KUKA KRL program: Machining3.src

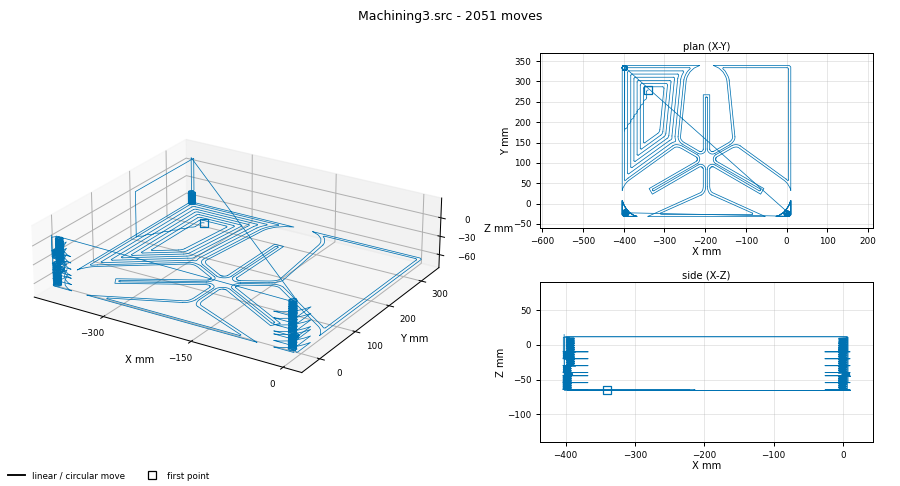
[picture p0: tool path of Machining3.src, 2051 of 2051 moves have a stored position in this frame; points joined in program order, loops and branches not executed]
&ACCESS RVP
&REL 1
&PARAM TEMPLATE = C:\KRC\Roboter\Template\vorgabe
&PARAM EDITMASK = *
DEF Machining3 ( )
LIN {X -339.907,Y 279.175,Z -64.500,A 0.015,B 0.000,C 180.000} C_DIS
CIRC {X -342.631,Y 278.046,Z -64.500,A 0.015,B -0.000,C -180.000},{X -343.760,Y 275.322,Z -64.500,A 0.015,B -0.000,C -180.000} C_DIS
LIN {X -343.759,Y 260.861,Z -64.500,A 0.015,B 0.000,C 180.000} C_DIS
CIRC {X -344.825,Y 257.341,Z -64.500,A 0.015,B 0.000,C 180.000},{X -347.664,Y 255.003,Z -64.500,A 0.015,B -0.000,C -180.000} C_DIS
CIRC {X -350.503,Y 252.666,Z -64.500,A 0.015,B 0.000,C 180.000},{X -351.569,Y 249.146,Z -64.500,A 0.015,B 0.000,C -180.000} C_DIS
LIN {X -351.566,Y 151.241,Z -64.500,A 0.015,B 0.000,C 180.000} C_DIS
CIRC {X -350.453,Y 149.418,Z -64.500,A 0.015,B 0.000,C -180.000},{X -348.323,Y 149.578,Z -64.500,A 0.015,B -0.000,C -180.000} C_DIS
LIN {X -316.688,Y 172.314,Z -64.500,A 0.015,B 0.000,C 180.000} C_DIS
CIRC {X -313.049,Y 176.334,Z -64.500,A 0.015,B 0.000,C 180.000},{X -311.385,Y 181.496,Z -64.500,A 0.015,B 0.000,C 180.000} C_DIS
LIN {X -301.199,Y 283.221,Z -64.500,A 0.015,B 0.000,C 180.000} C_DIS
CIRC {X -302.067,Y 285.859,Z -64.500,A 0.015,B 0.000,C 180.000},{X -304.605,Y 286.985,Z -64.500,A 0.015,B 0.000,C 180.000} C_DIS
LIN {X -347.717,Y 286.984,Z -64.500,A 0.015,B 0.000,C 180.000} C_DIS
CIRC {X -350.441,Y 285.856,Z -64.500,A 0.015,B 0.000,C 180.000},{X -351.570,Y 283.131,Z -64.500,A 0.015,B 0.000,C 180.000} C_DIS
LIN {X -351.569,Y 249.146,Z -64.500,A 0.015,B 0.000,C 180.000} C_DIS
CIRC {X -352.634,Y 245.626,Z -64.500,A 0.015,B 0.000,C 180.000},{X -355.473,Y 243.289,Z -64.500,A 0.015,B 0.000,C -180.000} C_DIS
CIRC {X -358.312,Y 240.951,Z -64.500,A 0.015,B 0.000,C 180.000},{X -359.378,Y 237.431,Z -64.500,A 0.015,B 0.000,C -180.000} C_DIS
LIN {X -359.375,Y 136.010,Z -64.500,A 0.015,B -0.000,C 180.000} C_DIS
CIRC {X -358.262,Y 134.188,Z -64.500,A 0.015,B 0.000,C 180.000},{X -356.132,Y 134.348,Z -64.500,A 0.015,B 0.000,C 180.000} C_DIS
LIN {X -309.268,Y 168.029,Z -64.500,A 0.015,B 0.000,C 180.000} C_DIS
CIRC {X -305.629,Y 172.049,Z -64.500,A 0.015,B 0.000,C -180.000},{X -303.966,Y 177.211,Z -64.500,A 0.015,B 0.000,C -180.000} C_DIS
LIN {X -292.568,Y 291.031,Z -64.500,A 0.015,B 0.000,C 180.000} C_DIS
CIRC {X -293.436,Y 293.669,Z -64.500,A 0.015,B -0.000,C -180.000},{X -295.974,Y 294.795,Z -64.500,A 0.015,B 0.000,C 180.000} C_DIS
LIN {X -355.527,Y 294.794,Z -64.500,A 0.015,B -0.000,C -180.000} C_DIS
CIRC {X -358.251,Y 293.665,Z -64.500,A 0.015,B 0.000,C -180.000},{X -359.380,Y 290.941,Z -64.500,A 0.015,B 0.000,C -180.000} C_DIS
LIN {X -359.378,Y 237.431,Z -64.500,A 0.015,B 0.000,C 180.000} C_DIS
CIRC {X -360.444,Y 233.911,Z -64.500,A 0.015,B 0.000,C 180.000},{X -363.283,Y 231.574,Z -64.500,A 0.015,B 0.000,C -180.000} C_DIS
CIRC {X -366.122,Y 229.236,Z -64.500,A 0.015,B 0.000,C -180.000},{X -367.188,Y 225.716,Z -64.500,A 0.015,B 0.000,C -180.000} C_DIS
LIN {X -367.185,Y 120.780,Z -64.500,A 0.015,B 0.000,C 180.000} C_DIS
CIRC {X -366.071,Y 118.958,Z -64.500,A 0.015,B -0.000,C 180.000},{X -363.942,Y 119.117,Z -64.500,A 0.015,B 0.000,C 180.000} C_DIS
LIN {X -301.848,Y 163.744,Z -64.500,A 0.015,B 0.000,C -180.000} C_DIS
CIRC {X -298.209,Y 167.764,Z -64.500,A 0.015,B 0.000,C 180.000},{X -296.546,Y 172.925,Z -64.500,A 0.015,B -0.000,C 180.000} C_DIS
LIN {X -283.937,Y 298.841,Z -64.500,A 0.015,B 0.000,C -180.000} C_DIS
CIRC {X -284.805,Y 301.479,Z -64.500,A 0.015,B 0.000,C 180.000},{X -287.343,Y 302.605,Z -64.500,A 0.015,B 0.000,C 180.000} C_DIS
LIN {X -363.337,Y 302.603,Z -64.500,A 0.015,B 0.000,C -180.000} C_DIS
CIRC {X -366.061,Y 301.475,Z -64.500,A 0.015,B 0.000,C 180.000},{X -367.190,Y 298.750,Z -64.500,A 0.015,B 0.000,C -180.000} C_DIS
LIN {X -367.188,Y 225.716,Z -64.500,A 0.015,B 0.000,C 180.000} C_DIS
CIRC {X -368.253,Y 222.196,Z -64.500,A 0.015,B 0.000,C -180.000},{X -371.092,Y 219.859,Z -64.500,A 0.015,B -0.000,C 180.000} C_DIS
CIRC {X -373.931,Y 217.521,Z -64.500,A 0.015,B -0.000,C 180.000},{X -374.997,Y 214.001,Z -64.500,A 0.015,B -0.000,C -180.000} C_DIS
LIN {X -374.994,Y 105.550,Z -64.500,A 0.015,B 0.000,C 180.000} C_DIS
CIRC {X -373.881,Y 103.728,Z -64.500,A 0.015,B 0.000,C 180.000},{X -371.751,Y 103.887,Z -64.500,A 0.015,B 0.000,C 180.000} C_DIS
LIN {X -293.623,Y 160.038,Z -64.500,A 0.015,B 0.000,C 180.000} C_DIS
CIRC {X -290.605,Y 163.373,Z -64.500,A 0.015,B 0.000,C 180.000},{X -289.225,Y 167.654,Z -64.500,A 0.015,B 0.000,C -180.000} C_DIS
LIN {X -275.691,Y 303.585,Z -64.500,A 0.015,B 0.000,C -180.000} C_DIS
CIRC {X -275.563,Y 304.401,Z -64.500,A 0.015,B 0.000,C -180.000},{X -275.412,Y 305.213,Z -64.500,A 0.015,B 0.000,C 180.000} C_DIS
CIRC {X -275.258,Y 306.024,Z -64.500,A 0.015,B 0.000,C 180.000},{X -275.124,Y 306.839,Z -64.500,A 0.015,B 0.000,C 180.000} C_DIS
CIRC {X -275.837,Y 309.333,Z -64.500,A 0.015,B 0.000,C 180.000},{X -278.194,Y 310.415,Z -64.500,A 0.015,B -0.000,C 180.000} C_DIS
LIN {X -371.147,Y 310.413,Z -64.500,A 0.015,B 0.000,C 180.000} C_DIS
CIRC {X -373.871,Y 309.285,Z -64.500,A 0.015,B -0.000,C 180.000},{X -375.000,Y 306.560,Z -64.500,A 0.015,B -0.000,C -180.000} C_DIS
LIN {X -374.997,Y 214.001,Z -64.500,A 0.015,B 0.000,C 180.000} C_DIS
CIRC {X -376.063,Y 210.481,Z -64.500,A 0.015,B 0.000,C -180.000},{X -378.902,Y 208.144,Z -64.500,A 0.015,B -0.000,C 180.000} C_DIS
CIRC {X -381.741,Y 205.806,Z -64.500,A 0.015,B 0.000,C -180.000},{X -382.807,Y 202.286,Z -64.500,A 0.015,B -0.000,C -180.000} C_DIS
LIN {X -382.803,Y 90.320,Z -64.500,A 0.015,B 0.000,C 180.000} C_DIS
CIRC {X -381.690,Y 88.498,Z -64.500,A 0.015,B -0.000,C -180.000},{X -379.561,Y 88.657,Z -64.500,A 0.015,B -0.000,C -180.000} C_DIS
LIN {X -288.345,Y 154.359,Z -64.500,A 0.015,B 0.000,C -180.000} C_DIS
CIRC {X -287.556,Y 154.885,Z -64.500,A 0.015,B 0.000,C 180.000},{X -286.733,Y 155.355,Z -64.500,A 0.015,B 0.000,C 180.000} C_DIS
CIRC {X -285.893,Y 155.792,Z -64.500,A 0.015,B 0.000,C 180.000},{X -285.049,Y 156.222,Z -64.500,A 0.015,B 0.000,C 180.000} C_DIS
CIRC {X -282.420,Y 158.717,Z -64.500,A 0.015,B -0.000,C 180.000},{X -281.597,Y 162.247,Z -64.500,A 0.015,B 0.000,C -180.000} C_DIS
CIRC {X -281.654,Y 163.235,Z -64.500,A 0.015,B 0.000,C -180.000},{X -281.701,Y 164.223,Z -64.500,A 0.015,B 0.000,C 180.000} C_DIS
CIRC {X -281.709,Y 165.212,Z -64.500,A 0.015,B 0.000,C -180.000},{X -281.645,Y 166.200,Z -64.500,A 0.015,B -0.000,C 180.000} C_DIS
LIN {X -267.342,Y 307.304,Z -64.500,A 0.015,B 0.000,C -180.000} C_DIS
CIRC {X -266.874,Y 309.190,Z -64.500,A 0.015,B 0.000,C 180.000},{X -266.314,Y 311.051,Z -64.500,A 0.015,B 0.000,C 180.000} C_DIS
CIRC {X -265.723,Y 312.902,Z -64.500,A 0.015,B -0.000,C 180.000},{X -265.158,Y 314.761,Z -64.500,A 0.015,B 0.000,C 180.000} C_DIS
CIRC {X -265.585,Y 317.142,Z -64.500,A 0.015,B -0.000,C 180.000},{X -267.747,Y 318.225,Z -64.500,A 0.015,B -0.000,C -180.000} C_DIS
LIN {X -378.957,Y 318.223,Z -64.500,A 0.015,B 0.000,C 180.000} C_DIS
CIRC {X -381.681,Y 317.094,Z -64.500,A 0.015,B 0.000,C 180.000},{X -382.810,Y 314.370,Z -64.500,A 0.015,B -0.000,C 180.000} C_DIS
LIN {X -382.807,Y 202.286,Z -64.500,A 0.015,B -0.000,C 180.000} C_DIS
CIRC {X -383.872,Y 198.767,Z -64.500,A 0.015,B 0.000,C 180.000},{X -386.711,Y 196.429,Z -64.500,A 0.015,B 0.000,C -180.000} C_DIS
CIRC {X -389.550,Y 194.091,Z -64.500,A 0.015,B -0.000,C 180.000},{X -390.616,Y 190.572,Z -64.500,A 0.015,B 0.000,C 180.000} C_DIS
LIN {X -390.613,Y 75.090,Z -64.500,A 0.015,B 0.000,C -180.000} C_DIS
CIRC {X -389.499,Y 73.268,Z -64.500,A 0.015,B -0.000,C -180.000},{X -387.370,Y 73.427,Z -64.500,A 0.015,B 0.000,C -180.000} C_DIS
LIN {X -283.893,Y 148.164,Z -64.500,A 0.015,B 0.000,C 180.000} C_DIS
CIRC {X -281.828,Y 149.430,Z -64.500,A 0.015,B 0.000,C 180.000},{X -279.602,Y 150.381,Z -64.500,A 0.015,B 0.000,C -180.000} C_DIS
CIRC {X -277.293,Y 151.093,Z -64.500,A 0.015,B 0.000,C 180.000},{X -274.944,Y 151.659,Z -64.500,A 0.015,B 0.000,C 180.000} C_DIS
CIRC {X -272.900,Y 153.122,Z -64.500,A 0.015,B 0.000,C 180.000},{X -272.606,Y 155.618,Z -64.500,A 0.015,B -0.000,C -180.000} C_DIS
CIRC {X -273.087,Y 157.304,Z -64.500,A 0.015,B 0.000,C -180.000},{X -273.496,Y 159.009,Z -64.500,A 0.015,B 0.000,C 180.000} C_DIS
CIRC {X -273.810,Y 160.735,Z -64.500,A 0.015,B 0.000,C 180.000},{X -274.004,Y 162.478,Z -64.500,A 0.015,B 0.000,C 180.000} C_DIS
CIRC {X -274.055,Y 163.218,Z -64.500,A 0.015,B 0.000,C -180.000},{X -274.097,Y 163.958,Z -64.500,A 0.015,B 0.000,C 180.000} C_DIS
CIRC {X -274.106,Y 164.700,Z -64.500,A 0.015,B 0.000,C -180.000},{X -274.060,Y 165.440,Z -64.500,A 0.015,B 0.000,C 180.000} C_DIS
LIN {X -260.011,Y 305.675,Z -64.500,A 0.015,B 0.000,C -180.000} C_DIS
CIRC {X -259.128,Y 309.215,Z -64.500,A 0.015,B 0.000,C 180.000},{X -258.064,Y 312.705,Z -64.500,A 0.015,B -0.000,C 180.000} C_DIS
CIRC {X -256.737,Y 316.107,Z -64.500,A 0.015,B 0.000,C 180.000},{X -255.075,Y 319.359,Z -64.500,A 0.015,B -0.000,C 180.000} C_DIS
CIRC {X -254.574,Y 320.199,Z -64.500,A 0.015,B 0.000,C -180.000},{X -254.046,Y 321.023,Z -64.500,A 0.015,B -0.000,C -180.000} C_DIS
CIRC {X -253.518,Y 321.847,Z -64.500,A 0.015,B 0.000,C 180.000},{X -253.017,Y 322.687,Z -64.500,A 0.015,B 0.000,C -180.000} C_DIS
CIRC {X -253.018,Y 324.920,Z -64.500,A 0.015,B 0.000,C 180.000},{X -254.952,Y 326.036,Z -64.500,A 0.015,B 0.000,C 180.000} C_DIS
LIN {X -386.767,Y 326.032,Z -64.500,A 0.015,B 0.000,C 180.000} C_DIS
CIRC {X -389.491,Y 324.904,Z -64.500,A 0.015,B 0.000,C 180.000},{X -390.620,Y 322.179,Z -64.500,A 0.015,B 0.000,C 180.000} C_DIS
LIN {X -390.616,Y 190.572,Z -64.500,A 0.015,B -0.000,C 180.000} C_DIS
CIRC {X -391.682,Y 187.052,Z -64.500,A 0.015,B 0.000,C -180.000},{X -394.521,Y 184.714,Z -64.500,A 0.015,B 0.000,C 180.000} C_DIS
CIRC {X -397.360,Y 182.376,Z -64.500,A 0.015,B 0.000,C -180.000},{X -398.426,Y 178.857,Z -64.500,A 0.015,B 0.000,C -180.000} C_DIS
LIN {X -398.422,Y 58.563,Z -64.500,A 0.015,B -0.000,C 180.000} C_DIS
CIRC {X -397.348,Y 56.920,Z -64.500,A 0.015,B 0.000,C -180.000},{X -395.413,Y 57.247,Z -64.500,A 0.015,B 0.000,C 180.000} C_DIS
CIRC {X -393.893,Y 58.674,Z -64.500,A 0.015,B 0.000,C 180.000},{X -392.395,Y 60.124,Z -64.500,A 0.015,B -0.000,C 180.000} C_DIS
CIRC {X -390.853,Y 61.528,Z -64.500,A 0.015,B 0.000,C 180.000},{X -389.207,Y 62.809,Z -64.500,A 0.015,B 0.000,C -180.000} C_DIS
LIN {X -279.477,Y 142.021,Z -64.500,A 0.015,B 0.000,C 180.000} C_DIS
CIRC {X -274.513,Y 144.373,Z -64.500,A 0.015,B 0.000,C 180.000},{X -269.038,Y 144.817,Z -64.500,A 0.015,B -0.000,C 180.000} C_DIS
CIRC {X -263.697,Y 143.918,Z -64.500,A 0.015,B 0.000,C 180.000},{X -258.524,Y 142.314,Z -64.500,A 0.015,B 0.000,C 180.000} C_DIS
CIRC {X -257.668,Y 141.957,Z -64.500,A 0.015,B 0.000,C 180.000},{X -256.832,Y 141.554,Z -64.500,A 0.015,B 0.000,C 180.000} C_DIS
CIRC {X -256.012,Y 141.120,Z -64.500,A 0.015,B 0.000,C -180.000},{X -255.203,Y 140.667,Z -64.500,A 0.015,B -0.000,C 180.000} C_DIS
LIN {X -219.429,Y 120.082,Z -64.500,A 0.015,B -0.000,C 180.000} C_DIS
CIRC {X -215.282,Y 116.094,Z -64.500,A 0.015,B -0.000,C 180.000},{X -213.463,Y 110.636,Z -64.500,A 0.015,B 0.000,C -180.000} C_DIS
CIRC {X -214.201,Y 104.972,Z -64.500,A 0.015,B 0.000,C 180.000},{X -217.183,Y 100.101,Z -64.500,A 0.015,B 0.000,C 180.000} C_DIS
CIRC {X -218.178,Y 99.193,Z -64.500,A 0.015,B 0.000,C -180.000},{X -219.295,Y 98.439,Z -64.500,A 0.015,B -0.000,C -180.000} C_DIS
LIN {X -328.516,Y 36.081,Z -64.500,A 0.015,B 0.000,C -180.000} C_DIS
CIRC {X -329.501,Y 34.796,Z -64.500,A 0.015,B -0.000,C -180.000},{X -329.289,Y 33.191,Z -64.500,A 0.015,B -0.000,C 180.000} C_DIS
LIN {X -328.854,Y 32.438,Z -64.500,A 0.015,B -0.000,C 180.000} C_DIS
CIRC {X -327.570,Y 31.454,Z -64.500,A 0.015,B 0.000,C -180.000},{X -325.966,Y 31.666,Z -64.500,A 0.015,B 0.000,C 180.000} C_DIS
LIN {X -217.356,Y 95.076,Z -64.500,A 0.015,B -0.000,C -180.000} C_DIS
CIRC {X -211.853,Y 96.649,Z -64.500,A 0.015,B 0.000,C 180.000},{X -206.257,Y 95.448,Z -64.500,A 0.015,B -0.000,C 180.000} C_DIS
CIRC {X -201.784,Y 91.960,Z -64.500,A 0.015,B 0.000,C -180.000},{X -199.085,Y 86.971,Z -64.500,A 0.015,B 0.000,C -180.000} C_DIS
CIRC {X -198.795,Y 85.656,Z -64.500,A 0.015,B 0.000,C 180.000},{X -198.698,Y 84.312,Z -64.500,A 0.015,B -0.000,C 180.000} C_DIS
LIN {X -199.059,Y 38.427,Z -64.500,A 0.015,B 0.000,C -180.000} C_DIS
CIRC {X -200.008,Y 33.666,Z -64.500,A 0.015,B 0.000,C -180.000},{X -201.868,Y 29.181,Z -64.500,A 0.015,B -0.000,C 180.000} C_DIS
CIRC {X -204.654,Y 25.192,Z -64.500,A 0.015,B 0.000,C -180.000},{X -208.294,Y 21.963,Z -64.500,A 0.015,B 0.000,C 180.000} C_DIS
CIRC {X -209.015,Y 21.509,Z -64.500,A 0.015,B 0.000,C -180.000},{X -209.775,Y 21.123,Z -64.500,A 0.015,B 0.000,C -180.000} C_DIS
LIN {X -309.427,Y -23.250,Z -64.500,A 0.015,B 0.000,C 180.000} C_DIS
CIRC {X -310.214,Y -24.810,Z -64.500,A 0.015,B 0.000,C -180.000},{X -308.854,Y -25.909,Z -64.500,A 0.015,B 0.000,C -180.000} C_DIS
LIN {X -84.669,Y -25.909,Z -64.500,A 0.015,B -0.000,C -180.000} C_DIS
CIRC {X -83.309,Y -24.810,Z -64.500,A 0.015,B -0.000,C -180.000},{X -84.096,Y -23.249,Z -64.500,A 0.015,B 0.000,C 180.000} C_DIS
LIN {X -183.958,Y 21.251,Z -64.500,A 0.015,B -0.000,C 180.000} C_DIS
CIRC {X -188.137,Y 24.080,Z -64.500,A 0.015,B 0.000,C 180.000},{X -191.126,Y 28.147,Z -64.500,A 0.015,B 0.000,C -180.000} C_DIS
CIRC {X -193.045,Y 32.747,Z -64.500,A 0.015,B 0.000,C 180.000},{X -194.326,Y 37.565,Z -64.500,A 0.015,B -0.000,C 180.000} C_DIS
CIRC {X -194.665,Y 39.888,Z -64.500,A 0.015,B 0.000,C 180.000},{X -194.784,Y 42.234,Z -64.500,A 0.015,B 0.000,C 180.000} C_DIS
LIN {X -194.814,Y 84.319,Z -64.500,A 0.015,B -0.000,C 180.000} C_DIS
CIRC {X -193.075,Y 90.605,Z -64.500,A 0.015,B 0.000,C 180.000},{X -188.354,Y 95.105,Z -64.500,A 0.015,B 0.000,C -180.000} C_DIS
CIRC {X -182.042,Y 96.633,Z -64.500,A 0.015,B 0.000,C 180.000},{X -175.783,Y 94.898,Z -64.500,A 0.015,B -0.000,C -180.000} C_DIS
LIN {X -67.545,Y 31.669,Z -64.500,A 0.015,B 0.000,C 180.000} C_DIS
CIRC {X -65.941,Y 31.456,Z -64.500,A 0.015,B 0.000,C -180.000},{X -64.657,Y 32.440,Z -64.500,A 0.015,B 0.000,C -180.000} C_DIS
LIN {X -64.222,Y 33.191,Z -64.500,A 0.015,B 0.000,C -180.000} C_DIS
CIRC {X -64.011,Y 34.796,Z -64.500,A 0.015,B 0.000,C 180.000},{X -64.996,Y 36.081,Z -64.500,A 0.015,B -0.000,C -180.000} C_DIS
LIN {X -174.232,Y 98.448,Z -64.500,A 0.015,B -0.000,C 180.000} C_DIS
CIRC {X -178.431,Y 102.562,Z -64.500,A 0.015,B 0.000,C -180.000},{X -180.120,Y 108.193,Z -64.500,A 0.015,B 0.000,C -180.000} C_DIS
CIRC {X -179.122,Y 113.930,Z -64.500,A 0.015,B -0.000,C 180.000},{X -175.856,Y 118.750,Z -64.500,A 0.015,B -0.000,C -180.000} C_DIS
CIRC {X -175.001,Y 119.475,Z -64.500,A 0.015,B 0.000,C -180.000},{X -174.065,Y 120.092,Z -64.500,A 0.015,B 0.000,C -180.000} C_DIS
LIN {X -133.766,Y 142.826,Z -64.500,A 0.015,B 0.000,C 180.000} C_DIS
CIRC {X -129.302,Y 144.292,Z -64.500,A 0.015,B -0.000,C 180.000},{X -124.636,Y 144.843,Z -64.500,A 0.015,B 0.000,C -180.000} C_DIS
CIRC {X -119.952,Y 144.386,Z -64.500,A 0.015,B 0.000,C 180.000},{X -115.494,Y 142.879,Z -64.500,A 0.015,B 0.000,C 180.000} C_DIS
CIRC {X -114.745,Y 142.483,Z -64.500,A 0.015,B 0.000,C 180.000},{X -114.035,Y 142.021,Z -64.500,A 0.015,B -0.000,C 180.000} C_DIS
LIN {X -1.197,Y 60.254,Z -64.500,A 0.015,B 0.000,C 180.000} C_DIS
CIRC {X -0.368,Y 59.547,Z -64.500,A 0.015,B -0.000,C 180.000},{X 0.396,Y 58.772,Z -64.500,A 0.015,B 0.000,C 180.000} C_DIS
CIRC {X 1.143,Y 57.981,Z -64.500,A 0.015,B -0.000,C -180.000},{X 1.925,Y 57.224,Z -64.500,A 0.015,B 0.000,C -180.000} C_DIS
CIRC {X 3.848,Y 56.900,Z -64.500,A 0.015,B 0.000,C -180.000},{X 4.916,Y 58.532,Z -64.500,A 0.015,B 0.000,C 180.000} C_DIS
LIN {X 4.908,Y 329.999,Z -64.500,A 0.015,B 0.000,C 180.000} C_DIS
CIRC {X 3.780,Y 332.723,Z -64.500,A 0.015,B 0.000,C -180.000},{X 1.055,Y 333.852,Z -64.500,A 0.015,B 0.000,C 180.000} C_DIS
LIN {X -155.007,Y 333.848,Z -64.500,A 0.015,B -0.000,C -180.000} C_DIS
CIRC {X -156.634,Y 332.740,Z -64.500,A 0.015,B 0.000,C 180.000},{X -156.200,Y 330.820,Z -64.500,A 0.015,B 0.000,C 180.000} C_DIS
CIRC {X -154.607,Y 329.358,Z -64.500,A 0.015,B 0.000,C 180.000},{X -152.990,Y 327.922,Z -64.500,A 0.015,B 0.000,C -180.000} C_DIS
CIRC {X -151.481,Y 326.364,Z -64.500,A 0.015,B 0.000,C 180.000},{X -150.250,Y 324.577,Z -64.500,A 0.015,B 0.000,C -180.000} C_DIS
CIRC {X -147.392,Y 319.491,Z -64.500,A 0.015,B 0.000,C 180.000},{X -144.610,Y 314.362,Z -64.500,A 0.015,B 0.000,C -180.000} C_DIS
CIRC {X -142.317,Y 308.973,Z -64.500,A 0.015,B 0.000,C -180.000},{X -140.995,Y 303.267,Z -64.500,A 0.015,B 0.000,C 180.000} C_DIS
LIN {X -126.980,Y 164.321,Z -64.500,A 0.015,B 0.000,C -180.000} C_DIS
CIRC {X -127.434,Y 158.876,Z -64.500,A 0.015,B 0.000,C -180.000},{X -129.803,Y 153.953,Z -64.500,A 0.015,B 0.000,C -180.000} C_DIS
CIRC {X -133.251,Y 149.818,Z -64.500,A 0.015,B 0.000,C 180.000},{X -137.197,Y 146.156,Z -64.500,A 0.015,B 0.000,C 180.000} C_DIS
CIRC {X -137.836,Y 145.658,Z -64.500,A 0.015,B 0.000,C 180.000},{X -138.496,Y 145.188,Z -64.500,A 0.015,B -0.000,C -180.000} C_DIS
CIRC {X -139.174,Y 144.745,Z -64.500,A 0.015,B 0.000,C 180.000},{X -139.868,Y 144.327,Z -64.500,A 0.015,B 0.000,C 180.000} C_DIS
LIN {X -176.147,Y 123.347,Z -64.500,A 0.015,B 0.000,C 180.000} C_DIS
CIRC {X -181.598,Y 121.768,Z -64.500,A 0.015,B 0.000,C 180.000},{X -187.157,Y 122.914,Z -64.500,A 0.015,B 0.000,C -180.000} C_DIS
CIRC {X -191.634,Y 126.325,Z -64.500,A 0.015,B 0.000,C -180.000},{X -194.376,Y 131.240,Z -64.500,A 0.015,B 0.000,C 180.000} C_DIS
CIRC {X -194.694,Y 132.613,Z -64.500,A 0.015,B 0.000,C -180.000},{X -194.801,Y 134.019,Z -64.500,A 0.015,B 0.000,C -180.000} C_DIS
LIN {X -194.206,Y 259.887,Z -64.500,A 0.015,B -0.000,C -180.000} C_DIS
CIRC {X -194.825,Y 261.382,Z -64.500,A 0.015,B -0.000,C 180.000},{X -196.320,Y 262.002,Z -64.500,A 0.015,B -0.000,C -180.000} C_DIS
LIN {X -197.192,Y 262.002,Z -64.500,A 0.015,B 0.000,C 180.000} C_DIS
CIRC {X -198.687,Y 261.382,Z -64.500,A 0.015,B 0.000,C 180.000},{X -199.306,Y 259.887,Z -64.500,A 0.015,B 0.000,C 180.000} C_DIS
LIN {X -198.711,Y 134.015,Z -64.500,A 0.015,B 0.000,C -180.000} C_DIS
CIRC {X -200.100,Y 128.501,Z -64.500,A 0.015,B -0.000,C 180.000},{X -203.935,Y 124.303,Z -64.500,A 0.015,B -0.000,C 180.000} C_DIS
CIRC {X -209.158,Y 122.206,Z -64.500,A 0.015,B 0.000,C 180.000},{X -214.785,Y 122.333,Z -64.500,A 0.015,B -0.000,C 180.000} C_DIS
CIRC {X -215.493,Y 122.525,Z -64.500,A 0.015,B -0.000,C 180.000},{X -216.182,Y 122.776,Z -64.500,A 0.015,B 0.000,C 180.000} C_DIS
CIRC {X -216.850,Y 123.077,Z -64.500,A 0.015,B 0.000,C -180.000},{X -217.497,Y 123.423,Z -64.500,A 0.015,B -0.000,C 180.000} C_DIS
LIN {X -256.621,Y 146.379,Z -64.500,A 0.015,B 0.000,C -180.000} C_DIS
CIRC {X -260.396,Y 149.649,Z -64.500,A 0.015,B 0.000,C 180.000},{X -263.446,Y 153.605,Z -64.500,A 0.015,B 0.000,C -180.000} C_DIS
CIRC {X -265.563,Y 158.141,Z -64.500,A 0.015,B -0.000,C -180.000},{X -266.540,Y 163.051,Z -64.500,A 0.015,B 0.000,C 180.000} C_DIS
CIRC {X -266.567,Y 163.869,Z -64.500,A 0.015,B 0.000,C 180.000},{X -266.521,Y 164.686,Z -64.500,A 0.015,B 0.000,C 180.000} C_DIS
LIN {X -252.387,Y 303.981,Z -64.500,A 0.015,B 0.000,C 180.000} C_DIS
CIRC {X -250.756,Y 309.943,Z -64.500,A 0.015,B -0.000,C 180.000},{X -248.557,Y 315.719,Z -64.500,A 0.015,B 0.000,C 180.000} C_DIS
CIRC {X -245.679,Y 321.198,Z -64.500,A 0.015,B -0.000,C 180.000},{X -242.052,Y 326.213,Z -64.500,A 0.015,B 0.000,C 180.000} C_DIS
CIRC {X -240.947,Y 327.442,Z -64.500,A 0.015,B 0.000,C 180.000},{X -239.759,Y 328.591,Z -64.500,A 0.015,B 0.000,C 180.000} C_DIS
CIRC {X -238.536,Y 329.702,Z -64.500,A 0.015,B -0.000,C -180.000},{X -237.321,Y 330.821,Z -64.500,A 0.015,B 0.000,C 180.000} C_DIS
CIRC {X -236.883,Y 332.738,Z -64.500,A 0.015,B 0.000,C -180.000},{X -238.508,Y 333.846,Z -64.500,A 0.015,B 0.000,C -180.000} C_DIS
LIN {X -394.577,Y 333.842,Z -64.500,A 0.015,B 0.000,C 180.000} C_DIS
CIRC {X -397.301,Y 332.713,Z -64.500,A 0.015,B -0.000,C -180.000},{X -398.430,Y 329.989,Z -64.500,A 0.015,B 0.000,C -180.000} C_DIS
LIN {X -398.426,Y 178.857,Z -64.500,A 0.015,B -0.000,C 180.000} C_DIS
LIN {X -398.270,Y 178.248,Z -64.330,A 0.015,B 0.000,C 180.000} C_DIS
LIN {X -397.978,Y 177.889,Z -63.865,A 0.015,B -0.000,C -180.000} C_DIS
LIN {X -397.842,Y 177.788,Z -63.230,A 0.015,B 0.000,C 180.000} C_DIS
$VEL.CP = 1.00000
LIN {X -397.842,Y 177.788,Z 11.000,A 0.015,B -0.000,C 180.000} C_DIS
$VEL.CP = 1.00000
LIN {X -397.447,Y 339.194,Z 11.000,A 0.015,B 0.000,C -180.000} C_DIS
$VEL.CP = 0.10000
LIN {X -397.447,Y 339.194,Z -42.731,A 0.015,B -0.000,C -180.000} C_DIS
LIN {X -397.509,Y 339.196,Z -43.123,A 0.015,B 0.000,C 180.000} C_DIS
LIN {X -397.689,Y 339.199,Z -43.477,A 0.015,B 0.000,C 180.000} C_DIS
LIN {X -398.507,Y 339.199,Z -43.983,A 0.015,B -0.000,C -180.000} C_DIS
LIN {X -398.672,Y 339.196,Z -44.000,A 0.015,B 0.000,C -180.000} C_DIS
LIN {X -399.336,Y 339.133,Z -44.023,A 0.015,B -0.000,C -180.000} C_DIS
LIN {X -399.552,Y 339.099,Z -44.031,A 0.015,B -0.000,C -180.000} C_DIS
LIN {X -402.866,Y 337.018,Z -44.171,A 0.015,B 0.000,C 180.000} C_DIS
LIN {X -402.887,Y 336.989,Z -44.173,A 0.015,B -0.000,C -180.000} C_DIS
LIN {X -403.357,Y 336.144,Z -44.206,A 0.015,B 0.000,C -180.000} C_DIS
LIN {X -403.418,Y 336.003,Z -44.212,A 0.015,B -0.000,C -180.000} C_DIS
LIN {X -403.598,Y 335.453,Z -44.232,A 0.015,B -0.000,C -180.000} C_DIS
LIN {X -403.636,Y 335.285,Z -44.238,A 0.015,B -0.000,C 180.000} C_DIS
LIN {X -403.753,Y 334.448,Z -44.268,A 0.015,B 0.000,C 180.000} C_DIS
LIN {X -403.779,Y 333.946,Z -44.285,A 0.015,B -0.000,C -180.000} C_DIS
LIN {X -403.787,Y 333.653,Z -44.295,A 0.015,B 0.000,C -180.000} C_DIS
LIN {X -403.787,Y 333.100,Z -44.315,A 0.015,B 0.000,C 180.000} C_DIS
LIN {X -401.273,Y 328.167,Z -44.515,A 0.015,B -0.000,C -180.000} C_DIS
LIN {X -395.804,Y 327.301,Z -44.716,A 0.015,B -0.000,C -180.000} C_DIS
LIN {X -391.889,Y 331.216,Z -44.917,A 0.015,B 0.000,C 180.000} C_DIS
LIN {X -392.755,Y 336.685,Z -45.117,A 0.015,B 0.000,C -180.000} C_DIS
LIN {X -397.689,Y 339.199,Z -45.318,A 0.015,B 0.000,C -180.000} C_DIS
LIN {X -398.507,Y 339.199,Z -45.347,A 0.015,B 0.000,C -180.000} C_DIS
LIN {X -399.336,Y 339.133,Z -45.376,A 0.015,B 0.000,C 180.000} C_DIS
LIN {X -399.552,Y 339.099,Z -45.384,A 0.015,B -0.000,C -180.000} C_DIS
LIN {X -402.866,Y 337.018,Z -45.524,A 0.015,B -0.000,C -180.000} C_DIS
LIN {X -402.887,Y 336.989,Z -45.525,A 0.015,B 0.000,C 180.000} C_DIS
LIN {X -403.357,Y 336.144,Z -45.559,A 0.015,B 0.000,C -180.000} C_DIS
LIN {X -403.418,Y 336.003,Z -45.564,A 0.015,B 0.000,C 180.000} C_DIS
LIN {X -403.598,Y 335.453,Z -45.585,A 0.015,B -0.000,C -180.000} C_DIS
LIN {X -403.636,Y 335.285,Z -45.591,A 0.015,B 0.000,C -180.000} C_DIS
LIN {X -403.753,Y 334.448,Z -45.620,A 0.015,B 0.000,C -180.000} C_DIS
LIN {X -403.779,Y 333.946,Z -45.638,A 0.015,B -0.000,C -180.000} C_DIS
LIN {X -403.787,Y 333.653,Z -45.648,A 0.015,B -0.000,C 180.000} C_DIS
LIN {X -403.787,Y 333.100,Z -45.667,A 0.015,B -0.000,C -180.000} C_DIS
LIN {X -401.273,Y 328.167,Z -45.868,A 0.015,B 0.000,C -180.000} C_DIS
LIN {X -395.804,Y 327.301,Z -46.069,A 0.015,B 0.000,C 180.000} C_DIS
LIN {X -391.889,Y 331.216,Z -46.269,A 0.015,B -0.000,C -180.000} C_DIS
LIN {X -392.755,Y 336.685,Z -46.470,A 0.015,B 0.000,C 180.000} C_DIS
LIN {X -397.689,Y 339.199,Z -46.671,A 0.015,B 0.000,C 180.000} C_DIS
LIN {X -398.507,Y 339.199,Z -46.699,A 0.015,B 0.000,C 180.000} C_DIS
LIN {X -399.336,Y 339.133,Z -46.728,A 0.015,B -0.000,C -180.000} C_DIS
LIN {X -399.552,Y 339.099,Z -46.736,A 0.015,B 0.000,C -180.000} C_DIS
LIN {X -402.866,Y 337.018,Z -46.876,A 0.015,B 0.000,C -180.000} C_DIS
LIN {X -402.887,Y 336.989,Z -46.878,A 0.015,B 0.000,C -180.000} C_DIS
LIN {X -403.357,Y 336.144,Z -46.912,A 0.015,B 0.000,C -180.000} C_DIS
LIN {X -403.418,Y 336.003,Z -46.917,A 0.015,B -0.000,C -180.000} C_DIS
LIN {X -403.598,Y 335.453,Z -46.937,A 0.015,B -0.000,C 180.000} C_DIS
LIN {X -403.636,Y 335.285,Z -46.943,A 0.015,B -0.000,C -180.000} C_DIS
LIN {X -403.753,Y 334.448,Z -46.973,A 0.015,B 0.000,C 180.000} C_DIS
LIN {X -403.779,Y 333.946,Z -46.990,A 0.015,B -0.000,C -180.000} C_DIS
LIN {X -403.787,Y 333.653,Z -47.000,A 0.015,B -0.000,C -180.000} C_DIS
LIN {X -403.787,Y 333.100,Z -47.020,A 0.015,B 0.000,C 180.000} C_DIS
LIN {X -401.273,Y 328.167,Z -47.220,A 0.015,B -0.000,C 180.000} C_DIS
LIN {X -395.804,Y 327.301,Z -47.421,A 0.015,B -0.000,C 180.000} C_DIS
LIN {X -391.889,Y 331.216,Z -47.622,A 0.015,B 0.000,C 180.000} C_DIS
LIN {X -392.755,Y 336.685,Z -47.823,A 0.015,B -0.000,C -180.000} C_DIS
LIN {X -397.689,Y 339.199,Z -48.023,A 0.015,B 0.000,C 180.000} C_DIS
LIN {X -398.507,Y 339.199,Z -48.052,A 0.015,B -0.000,C 180.000} C_DIS
LIN {X -399.336,Y 339.133,Z -48.081,A 0.015,B 0.000,C -180.000} C_DIS
LIN {X -399.552,Y 339.099,Z -48.089,A 0.015,B 0.000,C 180.000} C_DIS
LIN {X -402.866,Y 337.018,Z -48.229,A 0.015,B 0.000,C 180.000} C_DIS
LIN {X -402.887,Y 336.989,Z -48.230,A 0.015,B -0.000,C -180.000} C_DIS
LIN {X -403.357,Y 336.144,Z -48.264,A 0.015,B 0.000,C 180.000} C_DIS
LIN {X -403.418,Y 336.003,Z -48.269,A 0.015,B 0.000,C 180.000} C_DIS
LIN {X -403.598,Y 335.453,Z -48.290,A 0.015,B -0.000,C -180.000} C_DIS
LIN {X -403.636,Y 335.285,Z -48.296,A 0.015,B -0.000,C -180.000} C_DIS
LIN {X -403.753,Y 334.448,Z -48.325,A 0.015,B -0.000,C -180.000} C_DIS
LIN {X -403.779,Y 333.946,Z -48.343,A 0.015,B 0.000,C -180.000} C_DIS
LIN {X -403.787,Y 333.653,Z -48.353,A 0.015,B -0.000,C -180.000} C_DIS
LIN {X -403.787,Y 333.100,Z -48.372,A 0.015,B 0.000,C -180.000} C_DIS
LIN {X -401.273,Y 328.167,Z -48.573,A 0.015,B 0.000,C -180.000} C_DIS
LIN {X -395.804,Y 327.301,Z -48.774,A 0.015,B -0.000,C 180.000} C_DIS
LIN {X -391.889,Y 331.216,Z -48.974,A 0.015,B -0.000,C 180.000} C_DIS
LIN {X -392.755,Y 336.685,Z -49.175,A 0.015,B 0.000,C -180.000} C_DIS
LIN {X -397.689,Y 339.199,Z -49.376,A 0.015,B 0.000,C 180.000} C_DIS
LIN {X -398.507,Y 339.199,Z -49.404,A 0.015,B -0.000,C -180.000} C_DIS
LIN {X -399.336,Y 339.133,Z -49.433,A 0.015,B 0.000,C 180.000} C_DIS
LIN {X -399.552,Y 339.099,Z -49.441,A 0.015,B 0.000,C -180.000} C_DIS
LIN {X -402.866,Y 337.018,Z -49.582,A 0.015,B 0.000,C -180.000} C_DIS
LIN {X -402.887,Y 336.989,Z -49.583,A 0.015,B 0.000,C -180.000} C_DIS
LIN {X -403.357,Y 336.144,Z -49.617,A 0.015,B 0.000,C 180.000} C_DIS
LIN {X -403.418,Y 336.003,Z -49.622,A 0.015,B -0.000,C -180.000} C_DIS
LIN {X -403.598,Y 335.453,Z -49.642,A 0.015,B 0.000,C -180.000} C_DIS
LIN {X -403.636,Y 335.285,Z -49.648,A 0.015,B -0.000,C -180.000} C_DIS
LIN {X -403.753,Y 334.448,Z -49.678,A 0.015,B 0.000,C -180.000} C_DIS
LIN {X -403.779,Y 333.946,Z -49.695,A 0.015,B 0.000,C -180.000} C_DIS
LIN {X -403.787,Y 333.653,Z -49.706,A 0.015,B 0.000,C 180.000} C_DIS
LIN {X -403.787,Y 333.100,Z -49.725,A 0.015,B 0.000,C -180.000} C_DIS
LIN {X -401.273,Y 328.167,Z -49.926,A 0.015,B -0.000,C 180.000} C_DIS
LIN {X -395.804,Y 327.301,Z -50.126,A 0.015,B 0.000,C 180.000} C_DIS
LIN {X -391.889,Y 331.216,Z -50.327,A 0.015,B 0.000,C 180.000} C_DIS
LIN {X -392.755,Y 336.685,Z -50.528,A 0.015,B 0.000,C -180.000} C_DIS
LIN {X -397.689,Y 339.199,Z -50.728,A 0.015,B -0.000,C 180.000} C_DIS
LIN {X -398.507,Y 339.199,Z -50.757,A 0.015,B -0.000,C 180.000} C_DIS
LIN {X -399.336,Y 339.133,Z -50.786,A 0.015,B -0.000,C -180.000} C_DIS
LIN {X -399.552,Y 339.099,Z -50.794,A 0.015,B -0.000,C -180.000} C_DIS
LIN {X -402.866,Y 337.018,Z -50.934,A 0.015,B 0.000,C -180.000} C_DIS
LIN {X -402.887,Y 336.989,Z -50.935,A 0.015,B 0.000,C -180.000} C_DIS
LIN {X -403.357,Y 336.144,Z -50.969,A 0.015,B 0.000,C 180.000} C_DIS
LIN {X -403.418,Y 336.003,Z -50.975,A 0.015,B 0.000,C 180.000} C_DIS
LIN {X -403.598,Y 335.453,Z -50.995,A 0.015,B 0.000,C -180.000} C_DIS
LIN {X -403.636,Y 335.285,Z -51.001,A 0.015,B 0.000,C -180.000} C_DIS
LIN {X -403.753,Y 334.448,Z -51.030,A 0.015,B 0.000,C -180.000} C_DIS
LIN {X -403.779,Y 333.946,Z -51.048,A 0.015,B 0.000,C -180.000} C_DIS
LIN {X -403.787,Y 333.653,Z -51.058,A 0.015,B 0.000,C 180.000} C_DIS
LIN {X -403.787,Y 333.100,Z -51.077,A 0.015,B -0.000,C -180.000} C_DIS
LIN {X -401.273,Y 328.167,Z -51.278,A 0.015,B -0.000,C 180.000} C_DIS
LIN {X -395.804,Y 327.301,Z -51.479,A 0.015,B -0.000,C 180.000} C_DIS
LIN {X -391.889,Y 331.216,Z -51.680,A 0.015,B -0.000,C -180.000} C_DIS
LIN {X -392.755,Y 336.685,Z -51.880,A 0.015,B 0.000,C 180.000} C_DIS
LIN {X -397.689,Y 339.199,Z -52.081,A 0.015,B 0.000,C -180.000} C_DIS
LIN {X -398.507,Y 339.199,Z -52.110,A 0.015,B 0.000,C -180.000} C_DIS
LIN {X -399.336,Y 339.133,Z -52.139,A 0.015,B 0.000,C -180.000} C_DIS
LIN {X -399.552,Y 339.099,Z -52.146,A 0.015,B 0.000,C 180.000} C_DIS
LIN {X -402.866,Y 337.018,Z -52.287,A 0.015,B -0.000,C 180.000} C_DIS
LIN {X -402.887,Y 336.989,Z -52.288,A 0.015,B -0.000,C -180.000} C_DIS
LIN {X -403.357,Y 336.144,Z -52.322,A 0.015,B 0.000,C 180.000} C_DIS
LIN {X -403.418,Y 336.003,Z -52.327,A 0.015,B 0.000,C -180.000} C_DIS
LIN {X -403.598,Y 335.453,Z -52.347,A 0.015,B 0.000,C 180.000} C_DIS
LIN {X -403.636,Y 335.285,Z -52.353,A 0.015,B 0.000,C -180.000} C_DIS
LIN {X -403.753,Y 334.448,Z -52.383,A 0.015,B 0.000,C -180.000} C_DIS
LIN {X -403.779,Y 333.946,Z -52.400,A 0.015,B -0.000,C -180.000} C_DIS
LIN {X -403.787,Y 333.653,Z -52.411,A 0.015,B -0.000,C -180.000} C_DIS
LIN {X -403.787,Y 333.100,Z -52.430,A 0.015,B 0.000,C -180.000} C_DIS
LIN {X -401.273,Y 328.167,Z -52.631,A 0.015,B -0.000,C 180.000} C_DIS
LIN {X -395.804,Y 327.301,Z -52.831,A 0.015,B -0.000,C 180.000} C_DIS
LIN {X -391.889,Y 331.216,Z -53.032,A 0.015,B -0.000,C -180.000} C_DIS
LIN {X -392.755,Y 336.685,Z -53.233,A 0.015,B 0.000,C -180.000} C_DIS
LIN {X -397.689,Y 339.199,Z -53.433,A 0.015,B 0.000,C -180.000} C_DIS
LIN {X -398.507,Y 339.199,Z -53.462,A 0.015,B 0.000,C -180.000} C_DIS
LIN {X -399.336,Y 339.133,Z -53.491,A 0.015,B 0.000,C 180.000} C_DIS
LIN {X -399.552,Y 339.099,Z -53.499,A 0.015,B 0.000,C -180.000} C_DIS
LIN {X -402.866,Y 337.018,Z -53.639,A 0.015,B -0.000,C -180.000} C_DIS
LIN {X -402.887,Y 336.989,Z -53.640,A 0.015,B 0.000,C -180.000} C_DIS
LIN {X -403.357,Y 336.144,Z -53.674,A 0.015,B -0.000,C -180.000} C_DIS
LIN {X -403.418,Y 336.003,Z -53.680,A 0.015,B 0.000,C -180.000} C_DIS
LIN {X -403.598,Y 335.453,Z -53.700,A 0.015,B -0.000,C 180.000} C_DIS
LIN {X -403.636,Y 335.285,Z -53.706,A 0.015,B 0.000,C -180.000} C_DIS
LIN {X -403.753,Y 334.448,Z -53.735,A 0.015,B 0.000,C -180.000} C_DIS
LIN {X -403.779,Y 333.946,Z -53.753,A 0.015,B 0.000,C -180.000} C_DIS
LIN {X -403.787,Y 333.653,Z -53.763,A 0.015,B 0.000,C -180.000} C_DIS
LIN {X -403.787,Y 333.100,Z -53.783,A 0.015,B -0.000,C -180.000} C_DIS
LIN {X -401.273,Y 328.167,Z -53.983,A 0.015,B -0.000,C -180.000} C_DIS
LIN {X -395.804,Y 327.301,Z -54.184,A 0.015,B -0.000,C 180.000} C_DIS
LIN {X -391.889,Y 331.216,Z -54.385,A 0.015,B 0.000,C 180.000} C_DIS
LIN {X -392.755,Y 336.685,Z -54.585,A 0.015,B 0.000,C -180.000} C_DIS
LIN {X -397.689,Y 339.199,Z -54.786,A 0.015,B -0.000,C -180.000} C_DIS
LIN {X -398.507,Y 339.199,Z -54.815,A 0.015,B -0.000,C -180.000} C_DIS
LIN {X -399.336,Y 339.133,Z -54.844,A 0.015,B 0.000,C -180.000} C_DIS
LIN {X -399.552,Y 339.099,Z -54.851,A 0.015,B 0.000,C -180.000} C_DIS
LIN {X -402.866,Y 337.018,Z -54.992,A 0.015,B -0.000,C 180.000} C_DIS
LIN {X -402.887,Y 336.989,Z -54.993,A 0.015,B 0.000,C -180.000} C_DIS
LIN {X -403.357,Y 336.144,Z -55.027,A 0.015,B -0.000,C -180.000} C_DIS
LIN {X -403.418,Y 336.003,Z -55.032,A 0.015,B 0.000,C 180.000} C_DIS
LIN {X -403.598,Y 335.453,Z -55.052,A 0.015,B 0.000,C 180.000} C_DIS
LIN {X -403.636,Y 335.285,Z -55.058,A 0.015,B -0.000,C 180.000} C_DIS
LIN {X -403.753,Y 334.448,Z -55.088,A 0.015,B 0.000,C -180.000} C_DIS
LIN {X -403.779,Y 333.946,Z -55.105,A 0.015,B 0.000,C -180.000} C_DIS
LIN {X -403.787,Y 333.653,Z -55.116,A 0.015,B -0.000,C -180.000} C_DIS
LIN {X -403.787,Y 333.100,Z -55.135,A 0.015,B -0.000,C -180.000} C_DIS
LIN {X -401.273,Y 328.167,Z -55.336,A 0.015,B 0.000,C -180.000} C_DIS
LIN {X -395.804,Y 327.301,Z -55.536,A 0.015,B -0.000,C -180.000} C_DIS
LIN {X -391.889,Y 331.216,Z -55.737,A 0.015,B 0.000,C -180.000} C_DIS
LIN {X -392.755,Y 336.685,Z -55.938,A 0.015,B 0.000,C 180.000} C_DIS
LIN {X -397.689,Y 339.199,Z -56.139,A 0.015,B 0.000,C -180.000} C_DIS
LIN {X -398.507,Y 339.199,Z -56.167,A 0.015,B -0.000,C -180.000} C_DIS
LIN {X -399.336,Y 339.133,Z -56.196,A 0.015,B 0.000,C 180.000} C_DIS
LIN {X -399.552,Y 339.099,Z -56.204,A 0.015,B 0.000,C 180.000} C_DIS
LIN {X -402.866,Y 337.018,Z -56.344,A 0.015,B 0.000,C -180.000} C_DIS
LIN {X -402.887,Y 336.989,Z -56.346,A 0.015,B -0.000,C -180.000} C_DIS
LIN {X -403.357,Y 336.144,Z -56.379,A 0.015,B 0.000,C -180.000} C_DIS
LIN {X -403.418,Y 336.003,Z -56.385,A 0.015,B 0.000,C 180.000} C_DIS
LIN {X -403.598,Y 335.453,Z -56.405,A 0.015,B -0.000,C -180.000} C_DIS
LIN {X -403.636,Y 335.285,Z -56.411,A 0.015,B -0.000,C -180.000} C_DIS
LIN {X -403.753,Y 334.448,Z -56.441,A 0.015,B -0.000,C -180.000} C_DIS
LIN {X -403.779,Y 333.946,Z -56.458,A 0.015,B 0.000,C -180.000} C_DIS
LIN {X -403.787,Y 333.653,Z -56.468,A 0.015,B 0.000,C -180.000} C_DIS
LIN {X -403.787,Y 333.100,Z -56.488,A 0.015,B -0.000,C 180.000} C_DIS
LIN {X -401.273,Y 328.167,Z -56.688,A 0.015,B -0.000,C 180.000} C_DIS
LIN {X -395.804,Y 327.301,Z -56.889,A 0.015,B 0.000,C -180.000} C_DIS
LIN {X -391.889,Y 331.216,Z -57.090,A 0.015,B -0.000,C 180.000} C_DIS
LIN {X -392.755,Y 336.685,Z -57.290,A 0.015,B 0.000,C 180.000} C_DIS
LIN {X -397.689,Y 339.199,Z -57.491,A 0.015,B 0.000,C -180.000} C_DIS
LIN {X -398.507,Y 339.199,Z -57.520,A 0.015,B -0.000,C -180.000} C_DIS
LIN {X -399.336,Y 339.133,Z -57.549,A 0.015,B 0.000,C 180.000} C_DIS
LIN {X -399.552,Y 339.099,Z -57.556,A 0.015,B -0.000,C -180.000} C_DIS
LIN {X -402.866,Y 337.018,Z -57.697,A 0.015,B -0.000,C -180.000} C_DIS
LIN {X -402.887,Y 336.989,Z -57.698,A 0.015,B 0.000,C -180.000} C_DIS
LIN {X -403.357,Y 336.144,Z -57.732,A 0.015,B 0.000,C -180.000} C_DIS
LIN {X -403.418,Y 336.003,Z -57.737,A 0.015,B -0.000,C -180.000} C_DIS
LIN {X -403.598,Y 335.453,Z -57.758,A 0.015,B 0.000,C -180.000} C_DIS
LIN {X -403.636,Y 335.285,Z -57.764,A 0.015,B 0.000,C 180.000} C_DIS
LIN {X -403.753,Y 334.448,Z -57.793,A 0.015,B 0.000,C -180.000} C_DIS
LIN {X -403.779,Y 333.946,Z -57.811,A 0.015,B 0.000,C -180.000} C_DIS
LIN {X -403.787,Y 333.653,Z -57.821,A 0.015,B 0.000,C -180.000} C_DIS
LIN {X -403.787,Y 333.100,Z -57.840,A 0.015,B -0.000,C -180.000} C_DIS
LIN {X -401.273,Y 328.167,Z -58.041,A 0.015,B 0.000,C -180.000} C_DIS
LIN {X -395.804,Y 327.301,Z -58.242,A 0.015,B 0.000,C 180.000} C_DIS
LIN {X -391.889,Y 331.216,Z -58.442,A 0.015,B 0.000,C -180.000} C_DIS
LIN {X -392.755,Y 336.685,Z -58.643,A 0.015,B -0.000,C 180.000} C_DIS
LIN {X -397.689,Y 339.199,Z -58.844,A 0.015,B 0.000,C 180.000} C_DIS
LIN {X -398.507,Y 339.199,Z -58.872,A 0.015,B -0.000,C -180.000} C_DIS
LIN {X -399.336,Y 339.133,Z -58.901,A 0.015,B 0.000,C -180.000} C_DIS
LIN {X -399.552,Y 339.099,Z -58.909,A 0.015,B -0.000,C -180.000} C_DIS
LIN {X -402.866,Y 337.018,Z -59.049,A 0.015,B -0.000,C 180.000} C_DIS
LIN {X -402.887,Y 336.989,Z -59.051,A 0.015,B -0.000,C -180.000} C_DIS
LIN {X -403.357,Y 336.144,Z -59.084,A 0.015,B 0.000,C -180.000} C_DIS
LIN {X -403.418,Y 336.003,Z -59.090,A 0.015,B -0.000,C -180.000} C_DIS
LIN {X -403.598,Y 335.453,Z -59.110,A 0.015,B 0.000,C -180.000} C_DIS
LIN {X -403.636,Y 335.285,Z -59.116,A 0.015,B 0.000,C -180.000} C_DIS
LIN {X -403.753,Y 334.448,Z -59.146,A 0.015,B 0.000,C -180.000} C_DIS
LIN {X -403.779,Y 333.946,Z -59.163,A 0.015,B 0.000,C -180.000} C_DIS
LIN {X -403.787,Y 333.653,Z -59.173,A 0.015,B -0.000,C -180.000} C_DIS
LIN {X -403.787,Y 333.100,Z -59.193,A 0.015,B 0.000,C -180.000} C_DIS
LIN {X -401.273,Y 328.167,Z -59.393,A 0.015,B -0.000,C 180.000} C_DIS
LIN {X -395.804,Y 327.301,Z -59.594,A 0.015,B 0.000,C 180.000} C_DIS
LIN {X -391.889,Y 331.216,Z -59.795,A 0.015,B 0.000,C 180.000} C_DIS
LIN {X -392.755,Y 336.685,Z -59.996,A 0.015,B 0.000,C -180.000} C_DIS
LIN {X -397.689,Y 339.199,Z -60.196,A 0.015,B 0.000,C -180.000} C_DIS
LIN {X -398.507,Y 339.199,Z -60.225,A 0.015,B -0.000,C -180.000} C_DIS
LIN {X -399.336,Y 339.133,Z -60.254,A 0.015,B -0.000,C 180.000} C_DIS
LIN {X -399.552,Y 339.099,Z -60.262,A 0.015,B 0.000,C -180.000} C_DIS
LIN {X -402.866,Y 337.018,Z -60.402,A 0.015,B 0.000,C 180.000} C_DIS
LIN {X -402.887,Y 336.989,Z -60.403,A 0.015,B -0.000,C -180.000} C_DIS
LIN {X -403.357,Y 336.144,Z -60.437,A 0.015,B 0.000,C -180.000} C_DIS
LIN {X -403.418,Y 336.003,Z -60.442,A 0.015,B 0.000,C -180.000} C_DIS
LIN {X -403.598,Y 335.453,Z -60.463,A 0.015,B 0.000,C -180.000} C_DIS
LIN {X -403.636,Y 335.285,Z -60.469,A 0.015,B 0.000,C -180.000} C_DIS
LIN {X -403.753,Y 334.448,Z -60.498,A 0.015,B 0.000,C -180.000} C_DIS
LIN {X -403.779,Y 333.946,Z -60.516,A 0.015,B -0.000,C -180.000} C_DIS
LIN {X -403.787,Y 333.653,Z -60.526,A 0.015,B -0.000,C -180.000} C_DIS
LIN {X -403.787,Y 333.100,Z -60.545,A 0.015,B 0.000,C -180.000} C_DIS
LIN {X -401.273,Y 328.167,Z -60.746,A 0.015,B -0.000,C -180.000} C_DIS
LIN {X -395.804,Y 327.301,Z -60.947,A 0.015,B -0.000,C 180.000} C_DIS
LIN {X -391.889,Y 331.216,Z -61.147,A 0.015,B -0.000,C 180.000} C_DIS
LIN {X -392.755,Y 336.685,Z -61.348,A 0.015,B -0.000,C 180.000} C_DIS
LIN {X -397.689,Y 339.199,Z -61.549,A 0.015,B 0.000,C 180.000} C_DIS
LIN {X -398.507,Y 339.199,Z -61.577,A 0.015,B -0.000,C -180.000} C_DIS
LIN {X -399.336,Y 339.133,Z -61.606,A 0.015,B 0.000,C 180.000} C_DIS
LIN {X -399.552,Y 339.099,Z -61.614,A 0.015,B -0.000,C -180.000} C_DIS
LIN {X -402.866,Y 337.018,Z -61.754,A 0.015,B 0.000,C -180.000} C_DIS
LIN {X -402.887,Y 336.989,Z -61.756,A 0.015,B -0.000,C 180.000} C_DIS
LIN {X -403.357,Y 336.144,Z -61.790,A 0.015,B 0.000,C -180.000} C_DIS
LIN {X -403.418,Y 336.003,Z -61.795,A 0.015,B 0.000,C 180.000} C_DIS
LIN {X -403.598,Y 335.453,Z -61.815,A 0.015,B -0.000,C -180.000} C_DIS
LIN {X -403.636,Y 335.285,Z -61.821,A 0.015,B 0.000,C -180.000} C_DIS
LIN {X -403.753,Y 334.448,Z -61.851,A 0.015,B 0.000,C -180.000} C_DIS
LIN {X -403.779,Y 333.946,Z -61.868,A 0.015,B 0.000,C -180.000} C_DIS
LIN {X -403.787,Y 333.653,Z -61.878,A 0.015,B -0.000,C -180.000} C_DIS
LIN {X -403.787,Y 333.100,Z -61.898,A 0.015,B 0.000,C -180.000} C_DIS
LIN {X -401.273,Y 328.167,Z -62.098,A 0.015,B 0.000,C 180.000} C_DIS
LIN {X -395.804,Y 327.301,Z -62.299,A 0.015,B 0.000,C -180.000} C_DIS
LIN {X -391.889,Y 331.216,Z -62.500,A 0.015,B 0.000,C 180.000} C_DIS
LIN {X -392.755,Y 336.685,Z -62.701,A 0.015,B -0.000,C -180.000} C_DIS
LIN {X -397.689,Y 339.199,Z -62.901,A 0.015,B -0.000,C 180.000} C_DIS
LIN {X -398.507,Y 339.199,Z -62.930,A 0.015,B 0.000,C -180.000} C_DIS
LIN {X -399.336,Y 339.133,Z -62.959,A 0.015,B 0.000,C -180.000} C_DIS
LIN {X -399.552,Y 339.099,Z -62.967,A 0.015,B 0.000,C -180.000} C_DIS
LIN {X -402.866,Y 337.018,Z -63.107,A 0.015,B -0.000,C -180.000} C_DIS
LIN {X -402.887,Y 336.989,Z -63.108,A 0.015,B 0.000,C -180.000} C_DIS
LIN {X -403.357,Y 336.144,Z -63.142,A 0.015,B -0.000,C -180.000} C_DIS
LIN {X -403.418,Y 336.003,Z -63.147,A 0.015,B 0.000,C -180.000} C_DIS
LIN {X -403.598,Y 335.453,Z -63.168,A 0.015,B 0.000,C -180.000} C_DIS
LIN {X -403.636,Y 335.285,Z -63.174,A 0.015,B 0.000,C 180.000} C_DIS
LIN {X -403.753,Y 334.448,Z -63.203,A 0.015,B -0.000,C -180.000} C_DIS
LIN {X -403.779,Y 333.946,Z -63.221,A 0.015,B -0.000,C 180.000} C_DIS
LIN {X -403.787,Y 333.653,Z -63.231,A 0.015,B -0.000,C -180.000} C_DIS
LIN {X -403.787,Y 333.100,Z -63.250,A 0.015,B 0.000,C 180.000} C_DIS
LIN {X -401.273,Y 328.167,Z -63.451,A 0.015,B 0.000,C -180.000} C_DIS
LIN {X -395.804,Y 327.301,Z -63.652,A 0.015,B 0.000,C -180.000} C_DIS
LIN {X -391.889,Y 331.216,Z -63.852,A 0.015,B 0.000,C -180.000} C_DIS
LIN {X -392.755,Y 336.685,Z -64.053,A 0.015,B 0.000,C -180.000} C_DIS
LIN {X -397.689,Y 339.199,Z -64.254,A 0.015,B 0.000,C -180.000} C_DIS
LIN {X -398.507,Y 339.199,Z -64.282,A 0.015,B 0.000,C -180.000} C_DIS
LIN {X -399.336,Y 339.133,Z -64.312,A 0.015,B 0.000,C -180.000} C_DIS
LIN {X -399.552,Y 339.099,Z -64.319,A 0.015,B -0.000,C -180.000} C_DIS
LIN {X -402.866,Y 337.018,Z -64.460,A 0.015,B 0.000,C -180.000} C_DIS
LIN {X -402.887,Y 336.989,Z -64.461,A 0.015,B 0.000,C -180.000} C_DIS
LIN {X -403.357,Y 336.144,Z -64.495,A 0.015,B 0.000,C -180.000} C_DIS
LIN {X -403.418,Y 336.003,Z -64.500,A 0.015,B 0.000,C -180.000} C_DIS
LIN {X -403.533,Y 335.736,Z -64.500,A 0.015,B -0.000,C -180.000} C_DIS
LIN {X -403.730,Y 334.871,Z -64.500,A 0.015,B -0.000,C 180.000} C_DIS
LIN {X -403.787,Y 333.800,Z -64.500,A 0.015,B 0.000,C -180.000} C_DIS
LIN {X -403.779,Y 32.068,Z -64.500,A 0.015,B 0.000,C -180.000} C_DIS
LIN {X -402.839,Y 36.097,Z -64.500,A 0.015,B -0.000,C -180.000} C_DIS
LIN {X -402.682,Y 36.594,Z -64.500,A 0.015,B -0.000,C -180.000} C_DIS
LIN {X -401.989,Y 38.314,Z -64.500,A 0.015,B 0.000,C -180.000} C_DIS
LIN {X -401.777,Y 38.748,Z -64.500,A 0.015,B 0.000,C -180.000} C_DIS
LIN {X -396.446,Y 47.929,Z -64.500,A 0.015,B 0.000,C 180.000} C_DIS
LIN {X -396.102,Y 48.416,Z -64.500,A 0.015,B 0.000,C -180.000} C_DIS
LIN {X -393.338,Y 51.681,Z -64.500,A 0.015,B 0.000,C 180.000} C_DIS
LIN {X -393.237,Y 51.794,Z -64.500,A 0.015,B -0.000,C -180.000} C_DIS
LIN {X -392.240,Y 52.870,Z -64.500,A 0.015,B 0.000,C 180.000} C_DIS
LIN {X -392.056,Y 53.055,Z -64.500,A 0.015,B -0.000,C 180.000} C_DIS
LIN {X -389.153,Y 55.739,Z -64.500,A 0.015,B -0.000,C -180.000} C_DIS
LIN {X -388.927,Y 55.930,Z -64.500,A 0.015,B -0.000,C -180.000} C_DIS
LIN {X -386.025,Y 58.177,Z -64.500,A 0.015,B -0.000,C 180.000} C_DIS
LIN {X -385.929,Y 58.248,Z -64.500,A 0.015,B -0.000,C -180.000} C_DIS
LIN {X -276.034,Y 137.230,Z -64.500,A 0.015,B -0.000,C 180.000} C_DIS
LIN {X -275.463,Y 137.561,Z -64.500,A 0.015,B 0.000,C -180.000} C_DIS
LIN {X -273.618,Y 138.401,Z -64.500,A 0.015,B 0.000,C 180.000} C_DIS
LIN {X -272.904,Y 138.635,Z -64.500,A 0.015,B 0.000,C -180.000} C_DIS
LIN {X -271.453,Y 138.937,Z -64.500,A 0.015,B 0.000,C 180.000} C_DIS
LIN {X -270.894,Y 139.005,Z -64.500,A 0.015,B 0.000,C 180.000} C_DIS
LIN {X -269.443,Y 139.060,Z -64.500,A 0.015,B 0.000,C 180.000} C_DIS
LIN {X -268.903,Y 139.038,Z -64.500,A 0.015,B -0.000,C 180.000} C_DIS
LIN {X -266.726,Y 138.772,Z -64.500,A 0.015,B 0.000,C -180.000} C_DIS
LIN {X -266.283,Y 138.687,Z -64.500,A 0.015,B -0.000,C -180.000} C_DIS
LIN {X -264.106,Y 138.119,Z -64.500,A 0.015,B 0.000,C 180.000} C_DIS
LIN {X -263.744,Y 138.002,Z -64.500,A 0.015,B -0.000,C 180.000} C_DIS
LIN {X -260.646,Y 136.809,Z -64.500,A 0.015,B -0.000,C -180.000} C_DIS
LIN {X -260.330,Y 136.668,Z -64.500,A 0.015,B 0.000,C -180.000} C_DIS
LIN {X -258.301,Y 135.637,Z -64.500,A 0.015,B -0.000,C 180.000} C_DIS
LIN {X -258.145,Y 135.553,Z -64.500,A 0.015,B 0.000,C 180.000} C_DIS
LIN {X -222.389,Y 114.978,Z -64.500,A 0.015,B 0.000,C -180.000} C_DIS
LIN {X -221.736,Y 114.489,Z -64.500,A 0.015,B 0.000,C 180.000} C_DIS
LIN {X -220.980,Y 113.765,Z -64.500,A 0.015,B 0.000,C 180.000} C_DIS
CIRC {X -220.643,Y 113.390,Z -64.500,A 0.015,B 0.000,C 180.000},{X -220.366,Y 112.970,Z -64.500,A 0.015,B -0.000,C 180.000} C_DIS
LIN {X -219.872,Y 112.084,Z -64.500,A 0.015,B 0.000,C -180.000} C_DIS
CIRC {X -219.654,Y 111.612,Z -64.500,A 0.015,B 0.000,C 180.000},{X -219.512,Y 111.113,Z -64.500,A 0.015,B -0.000,C 180.000} C_DIS
LIN {X -219.290,Y 110.024,Z -64.500,A 0.015,B 0.000,C 180.000} C_DIS
CIRC {X -219.224,Y 109.489,Z -64.500,A 0.015,B 0.000,C -180.000},{X -219.245,Y 108.949,Z -64.500,A 0.015,B 0.000,C 180.000} C_DIS
LIN {X -219.375,Y 107.861,Z -64.500,A 0.015,B 0.000,C -180.000} C_DIS
CIRC {X -219.485,Y 107.317,Z -64.500,A 0.015,B -0.000,C 180.000},{X -219.683,Y 106.799,Z -64.500,A 0.015,B 0.000,C 180.000} C_DIS
LIN {X -220.189,Y 105.742,Z -64.500,A 0.015,B 0.000,C 180.000} C_DIS
CIRC {X -220.453,Y 105.286,Z -64.500,A 0.015,B 0.000,C -180.000},{X -220.786,Y 104.876,Z -64.500,A 0.015,B -0.000,C 180.000} C_DIS
LIN {X -221.463,Y 104.161,Z -64.500,A 0.015,B 0.000,C 180.000} C_DIS
LIN {X -222.227,Y 103.559,Z -64.500,A 0.015,B 0.000,C 180.000} C_DIS
LIN {X -337.671,Y 36.985,Z -64.500,A 0.015,B 0.000,C -180.000} C_DIS
LIN {X -329.752,Y 23.290,Z -64.500,A 0.015,B 0.000,C -180.000} C_DIS
LIN {X -214.411,Y 89.964,Z -64.500,A 0.015,B 0.000,C -180.000} C_DIS
LIN {X -213.533,Y 90.318,Z -64.500,A 0.015,B 0.000,C -180.000} C_DIS
LIN {X -212.574,Y 90.556,Z -64.500,A 0.015,B 0.000,C 180.000} C_DIS
LIN {X -211.588,Y 90.651,Z -64.500,A 0.015,B 0.000,C 180.000} C_DIS
LIN {X -210.548,Y 90.599,Z -64.500,A 0.015,B 0.000,C 180.000} C_DIS
LIN {X -209.592,Y 90.410,Z -64.500,A 0.015,B 0.000,C 180.000} C_DIS
LIN {X -208.689,Y 90.091,Z -64.500,A 0.015,B 0.000,C 180.000} C_DIS
CIRC {X -208.223,Y 89.885,Z -64.500,A 0.015,B 0.000,C -180.000},{X -207.792,Y 89.612,Z -64.500,A 0.015,B 0.000,C 180.000} C_DIS
LIN {X -206.889,Y 88.937,Z -64.500,A 0.015,B 0.000,C -180.000} C_DIS
CIRC {X -206.473,Y 88.570,Z -64.500,A 0.015,B -0.000,C 180.000},{X -206.123,Y 88.140,Z -64.500,A 0.015,B 0.000,C 180.000} C_DIS
LIN {X -205.479,Y 87.200,Z -64.500,A 0.015,B -0.000,C 180.000} C_DIS
CIRC {X -205.217,Y 86.744,Z -64.500,A 0.015,B 0.000,C 180.000},{X -205.028,Y 86.254,Z -64.500,A 0.015,B 0.000,C 180.000} C_DIS
LIN {X -204.739,Y 85.285,Z -64.500,A 0.015,B -0.000,C 180.000} C_DIS
LIN {X -204.598,Y 84.317,Z -64.500,A 0.015,B 0.000,C 180.000} C_DIS
LIN {X -204.628,Y 42.238,Z -64.500,A 0.015,B -0.000,C -180.000} C_DIS
LIN {X -204.645,Y 41.908,Z -64.500,A 0.015,B 0.000,C 180.000} C_DIS
LIN {X -204.931,Y 39.006,Z -64.500,A 0.015,B 0.000,C -180.000} C_DIS
LIN {X -204.977,Y 38.692,Z -64.500,A 0.015,B -0.000,C -180.000} C_DIS
LIN {X -205.542,Y 35.790,Z -64.500,A 0.015,B -0.000,C 180.000} C_DIS
LIN {X -205.632,Y 35.431,Z -64.500,A 0.015,B 0.000,C 180.000} C_DIS
LIN {X -206.084,Y 33.980,Z -64.500,A 0.015,B 0.000,C 180.000} C_DIS
LIN {X -206.215,Y 33.628,Z -64.500,A 0.015,B 0.000,C 180.000} C_DIS
LIN {X -207.108,Y 31.590,Z -64.500,A 0.015,B 0.000,C 180.000} C_DIS
LIN {X -207.434,Y 31.010,Z -64.500,A 0.015,B -0.000,C 180.000} C_DIS
LIN {X -208.443,Y 29.566,Z -64.500,A 0.015,B -0.000,C 180.000} C_DIS
LIN {X -208.778,Y 29.158,Z -64.500,A 0.015,B 0.000,C -180.000} C_DIS
LIN {X -209.548,Y 28.357,Z -64.500,A 0.015,B 0.000,C 180.000} C_DIS
LIN {X -210.055,Y 27.925,Z -64.500,A 0.015,B 0.000,C 180.000} C_DIS
LIN {X -211.662,Y 26.807,Z -64.500,A 0.015,B -0.000,C 180.000} C_DIS
LIN {X -212.202,Y 26.501,Z -64.500,A 0.015,B 0.000,C 180.000} C_DIS
LIN {X -336.127,Y -29.421,Z -64.500,A 0.015,B 0.000,C 180.000} C_DIS
LIN {X -336.254,Y -29.475,Z -64.500,A 0.015,B 0.000,C 180.000} C_DIS
LIN {X -339.156,Y -30.644,Z -64.500,A 0.015,B 0.000,C 180.000} C_DIS
LIN {X -339.405,Y -30.734,Z -64.500,A 0.015,B -0.000,C 180.000} C_DIS
LIN {X -341.098,Y -31.266,Z -64.500,A 0.015,B -0.000,C 180.000} C_DIS
LIN {X -52.414,Y -31.266,Z -64.500,A 0.015,B -0.000,C 180.000} C_DIS
LIN {X -54.106,Y -30.734,Z -64.500,A 0.015,B 0.000,C -180.000} C_DIS
LIN {X -54.377,Y -30.636,Z -64.500,A 0.015,B -0.000,C -180.000} C_DIS
LIN {X -58.153,Y -29.085,Z -64.500,A 0.015,B 0.000,C -180.000} C_DIS
LIN {X -58.260,Y -29.039,Z -64.500,A 0.015,B 0.000,C -180.000} C_DIS
LIN {X -181.529,Y 26.628,Z -64.500,A 0.015,B -0.000,C 180.000} C_DIS
LIN {X -182.152,Y 26.994,Z -64.500,A 0.015,B -0.000,C 180.000} C_DIS
LIN {X -183.786,Y 28.206,Z -64.500,A 0.015,B 0.000,C 180.000} C_DIS
LIN {X -184.358,Y 28.744,Z -64.500,A 0.015,B 0.000,C -180.000} C_DIS
LIN {X -185.335,Y 29.905,Z -64.500,A 0.015,B 0.000,C -180.000} C_DIS
LIN {X -185.667,Y 30.375,Z -64.500,A 0.015,B 0.000,C -180.000} C_DIS
LIN {X -186.433,Y 31.684,Z -64.500,A 0.015,B -0.000,C 180.000} C_DIS
LIN {X -186.621,Y 32.056,Z -64.500,A 0.015,B 0.000,C -180.000} C_DIS
LIN {X -187.306,Y 33.649,Z -64.500,A 0.015,B -0.000,C -180.000} C_DIS
LIN {X -187.428,Y 33.980,Z -64.500,A 0.015,B -0.000,C -180.000} C_DIS
LIN {X -187.880,Y 35.431,Z -64.500,A 0.015,B 0.000,C -180.000} C_DIS
LIN {X -187.970,Y 35.790,Z -64.500,A 0.015,B 0.000,C -180.000} C_DIS
LIN {X -188.535,Y 38.692,Z -64.500,A 0.015,B 0.000,C -180.000} C_DIS
LIN {X -188.581,Y 39.006,Z -64.500,A 0.015,B 0.000,C -180.000} C_DIS
LIN {X -188.867,Y 41.908,Z -64.500,A 0.015,B -0.000,C 180.000} C_DIS
LIN {X -188.884,Y 42.238,Z -64.500,A 0.015,B -0.000,C 180.000} C_DIS
LIN {X -188.914,Y 84.317,Z -64.500,A 0.015,B 0.000,C 180.000} C_DIS
LIN {X -188.773,Y 85.285,Z -64.500,A 0.015,B 0.000,C -180.000} C_DIS
LIN {X -188.484,Y 86.254,Z -64.500,A 0.015,B -0.000,C 180.000} C_DIS
CIRC {X -188.295,Y 86.744,Z -64.500,A 0.015,B -0.000,C 180.000},{X -188.033,Y 87.200,Z -64.500,A 0.015,B 0.000,C -180.000} C_DIS
LIN {X -187.388,Y 88.140,Z -64.500,A 0.015,B -0.000,C 180.000} C_DIS
LIN {X -186.934,Y 88.674,Z -64.500,A 0.015,B 0.000,C -180.000} C_DIS
LIN {X -186.718,Y 88.880,Z -64.500,A 0.015,B 0.000,C 180.000} C_DIS
LIN {X -186.187,Y 89.294,Z -64.500,A 0.015,B 0.000,C -180.000} C_DIS
LIN {X -185.274,Y 89.870,Z -64.500,A 0.015,B 0.000,C -180.000} C_DIS
CIRC {X -184.812,Y 90.113,Z -64.500,A 0.015,B 0.000,C -180.000},{X -184.317,Y 90.283,Z -64.500,A 0.015,B 0.000,C 180.000} C_DIS
LIN {X -183.294,Y 90.548,Z -64.500,A 0.015,B 0.000,C -180.000} C_DIS
CIRC {X -182.788,Y 90.638,Z -64.500,A 0.015,B 0.000,C -180.000},{X -182.275,Y 90.651,Z -64.500,A 0.015,B 0.000,C 180.000} C_DIS
LIN {X -181.235,Y 90.599,Z -64.500,A 0.015,B -0.000,C 180.000} C_DIS
CIRC {X -180.730,Y 90.535,Z -64.500,A 0.015,B -0.000,C -180.000},{X -180.241,Y 90.396,Z -64.500,A 0.015,B 0.000,C -180.000} C_DIS
LIN {X -179.265,Y 90.038,Z -64.500,A 0.015,B 0.000,C 180.000} C_DIS
LIN {X -178.737,Y 89.791,Z -64.500,A 0.015,B 0.000,C -180.000} C_DIS
LIN {X -63.759,Y 23.290,Z -64.500,A 0.015,B -0.000,C 180.000} C_DIS
LIN {X -55.841,Y 36.985,Z -64.500,A 0.015,B 0.000,C 180.000} C_DIS
LIN {X -171.285,Y 103.559,Z -64.500,A 0.015,B -0.000,C 180.000} C_DIS
LIN {X -172.049,Y 104.161,Z -64.500,A 0.015,B 0.000,C -180.000} C_DIS
LIN {X -172.726,Y 104.876,Z -64.500,A 0.015,B -0.000,C -180.000} C_DIS
CIRC {X -173.058,Y 105.286,Z -64.500,A 0.015,B 0.000,C -180.000},{X -173.323,Y 105.742,Z -64.500,A 0.015,B 0.000,C 180.000} C_DIS
LIN {X -173.829,Y 106.799,Z -64.500,A 0.015,B -0.000,C 180.000} C_DIS
CIRC {X -174.027,Y 107.317,Z -64.500,A 0.015,B -0.000,C -180.000},{X -174.137,Y 107.861,Z -64.500,A 0.015,B 0.000,C 180.000} C_DIS
LIN {X -174.267,Y 108.949,Z -64.500,A 0.015,B -0.000,C -180.000} C_DIS
CIRC {X -174.287,Y 109.489,Z -64.500,A 0.015,B 0.000,C -180.000},{X -174.222,Y 110.024,Z -64.500,A 0.015,B 0.000,C -180.000} C_DIS
LIN {X -174.000,Y 111.113,Z -64.500,A 0.015,B 0.000,C -180.000} C_DIS
CIRC {X -173.858,Y 111.612,Z -64.500,A 0.015,B 0.000,C -180.000},{X -173.640,Y 112.084,Z -64.500,A 0.015,B 0.000,C 180.000} C_DIS
LIN {X -173.146,Y 112.970,Z -64.500,A 0.015,B -0.000,C 180.000} C_DIS
CIRC {X -172.869,Y 113.390,Z -64.500,A 0.015,B 0.000,C -180.000},{X -172.532,Y 113.765,Z -64.500,A 0.015,B 0.000,C -180.000} C_DIS
LIN {X -171.775,Y 114.489,Z -64.500,A 0.015,B 0.000,C -180.000} C_DIS
LIN {X -171.123,Y 114.978,Z -64.500,A 0.015,B 0.000,C -180.000} C_DIS
LIN {X -134.690,Y 135.941,Z -64.500,A 0.015,B 0.000,C -180.000} C_DIS
LIN {X -134.374,Y 136.102,Z -64.500,A 0.015,B -0.000,C -180.000} C_DIS
LIN {X -131.374,Y 137.432,Z -64.500,A 0.015,B 0.000,C 180.000} C_DIS
LIN {X -131.117,Y 137.534,Z -64.500,A 0.015,B 0.000,C 180.000} C_DIS
LIN {X -129.666,Y 138.040,Z -64.500,A 0.015,B 0.000,C -180.000} C_DIS
LIN {X -129.405,Y 138.119,Z -64.500,A 0.015,B 0.000,C 180.000} C_DIS
LIN {X -127.229,Y 138.687,Z -64.500,A 0.015,B 0.000,C 180.000} C_DIS
LIN {X -126.741,Y 138.777,Z -64.500,A 0.015,B 0.000,C 180.000} C_DIS
LIN {X -124.202,Y 139.053,Z -64.500,A 0.015,B -0.000,C 180.000} C_DIS
LIN {X -123.558,Y 139.062,Z -64.500,A 0.015,B 0.000,C 180.000} C_DIS
LIN {X -122.106,Y 138.942,Z -64.500,A 0.015,B 0.000,C 180.000} C_DIS
LIN {X -121.507,Y 138.838,Z -64.500,A 0.015,B -0.000,C 180.000} C_DIS
LIN {X -120.056,Y 138.448,Z -64.500,A 0.015,B 0.000,C -180.000} C_DIS
LIN {X -119.491,Y 138.241,Z -64.500,A 0.015,B -0.000,C 180.000} C_DIS
LIN {X -118.010,Y 137.542,Z -64.500,A 0.015,B 0.000,C -180.000} C_DIS
LIN {X -117.478,Y 137.230,Z -64.500,A 0.015,B -0.000,C 180.000} C_DIS
LIN {X -7.301,Y 58.046,Z -64.500,A 0.015,B 0.000,C -180.000} C_DIS
LIN {X -7.195,Y 57.966,Z -64.500,A 0.015,B 0.000,C -180.000} C_DIS
LIN {X -4.575,Y 55.923,Z -64.500,A 0.015,B 0.000,C -180.000} C_DIS
LIN {X -4.359,Y 55.739,Z -64.500,A 0.015,B 0.000,C 180.000} C_DIS
LIN {X -1.456,Y 53.055,Z -64.500,A 0.015,B -0.000,C 180.000} C_DIS
LIN {X -1.210,Y 52.802,Z -64.500,A 0.015,B 0.000,C -180.000} C_DIS
LIN {X 2.280,Y 48.824,Z -64.500,A 0.015,B 0.000,C 180.000} C_DIS
LIN {X 2.639,Y 48.332,Z -64.500,A 0.015,B 0.000,C 180.000} C_DIS
LIN {X 4.953,Y 44.470,Z -64.500,A 0.015,B 0.000,C 180.000} C_DIS
LIN {X 4.979,Y 44.426,Z -64.500,A 0.015,B -0.000,C 180.000} C_DIS
LIN {X 8.268,Y 38.744,Z -64.500,A 0.015,B -0.000,C -180.000} C_DIS
LIN {X 8.490,Y 38.281,Z -64.500,A 0.015,B -0.000,C -180.000} C_DIS
LIN {X 9.297,Y 36.217,Z -64.500,A 0.015,B 0.000,C 180.000} C_DIS
LIN {X 9.445,Y 35.738,Z -64.500,A 0.015,B 0.000,C 180.000} C_DIS
LIN {X 10.273,Y 32.108,Z -64.500,A 0.015,B 0.000,C 180.000} C_DIS
LIN {X 10.265,Y 334.347,Z -64.500,A 0.015,B 0.000,C -180.000} C_DIS
LIN {X 10.072,Y 335.556,Z -64.500,A 0.015,B 0.000,C 180.000} C_DIS
LIN {X 9.898,Y 336.018,Z -64.500,A 0.015,B 0.000,C 180.000} C_DIS
LIN {X 9.664,Y 336.377,Z -64.500,A 0.015,B 0.000,C 180.000} C_DIS
LIN {X 7.374,Y 338.634,Z -64.500,A 0.015,B -0.000,C -180.000} C_DIS
LIN {X 7.069,Y 338.840,Z -64.500,A 0.015,B -0.000,C -180.000} C_DIS
LIN {X 6.802,Y 338.955,Z -64.500,A 0.015,B -0.000,C 180.000} C_DIS
LIN {X 5.937,Y 339.152,Z -64.500,A 0.015,B -0.000,C 180.000} C_DIS
LIN {X 4.865,Y 339.209,Z -64.500,A 0.015,B -0.000,C 180.000} C_DIS
LIN {X -180.113,Y 339.204,Z -64.500,A 0.015,B -0.000,C -180.000} C_DIS
LIN {X -179.927,Y 339.176,Z -64.500,A 0.015,B 0.000,C 180.000} C_DIS
LIN {X -179.331,Y 339.030,Z -64.500,A 0.015,B 0.000,C -180.000} C_DIS
LIN {X -178.242,Y 338.656,Z -64.500,A 0.015,B 0.000,C 180.000} C_DIS
LIN {X -177.868,Y 338.501,Z -64.500,A 0.015,B 0.000,C 180.000} C_DIS
LIN {X -167.347,Y 333.405,Z -64.500,A 0.015,B 0.000,C 180.000} C_DIS
LIN {X -166.810,Y 333.080,Z -64.500,A 0.015,B 0.000,C 180.000} C_DIS
LIN {X -165.359,Y 332.006,Z -64.500,A 0.015,B 0.000,C -180.000} C_DIS
LIN {X -165.063,Y 331.761,Z -64.500,A 0.015,B -0.000,C 180.000} C_DIS
LIN {X -157.163,Y 324.392,Z -64.500,A 0.015,B 0.000,C -180.000} C_DIS
LIN {X -156.792,Y 323.986,Z -64.500,A 0.015,B 0.000,C 180.000} C_DIS
LIN {X -155.392,Y 322.172,Z -64.500,A 0.015,B 0.000,C -180.000} C_DIS
LIN {X -155.133,Y 321.784,Z -64.500,A 0.015,B 0.000,C -180.000} C_DIS
LIN {X -149.946,Y 312.715,Z -64.500,A 0.015,B 0.000,C -180.000} C_DIS
LIN {X -149.707,Y 312.201,Z -64.500,A 0.015,B -0.000,C 180.000} C_DIS
LIN {X -148.509,Y 308.936,Z -64.500,A 0.015,B 0.000,C 180.000} C_DIS
LIN {X -148.440,Y 308.726,Z -64.500,A 0.015,B -0.000,C 180.000} C_DIS
LIN {X -147.586,Y 305.824,Z -64.500,A 0.015,B -0.000,C -180.000} C_DIS
LIN {X -147.529,Y 305.603,Z -64.500,A 0.015,B 0.000,C 180.000} C_DIS
LIN {X -146.884,Y 302.701,Z -64.500,A 0.015,B -0.000,C -180.000} C_DIS
LIN {X -146.837,Y 302.441,Z -64.500,A 0.015,B 0.000,C -180.000} C_DIS
LIN {X -146.426,Y 299.539,Z -64.500,A 0.015,B -0.000,C 180.000} C_DIS
LIN {X -146.410,Y 299.402,Z -64.500,A 0.015,B 0.000,C 180.000} C_DIS
LIN {X -132.851,Y 163.734,Z -64.500,A 0.015,B 0.000,C -180.000} C_DIS
LIN {X -132.859,Y 162.990,Z -64.500,A 0.015,B 0.000,C -180.000} C_DIS
LIN {X -133.123,Y 160.814,Z -64.500,A 0.015,B 0.000,C 180.000} C_DIS
LIN {X -133.320,Y 160.018,Z -64.500,A 0.015,B -0.000,C -180.000} C_DIS
LIN {X -133.873,Y 158.567,Z -64.500,A 0.015,B 0.000,C 180.000} C_DIS
LIN {X -134.078,Y 158.126,Z -64.500,A 0.015,B 0.000,C -180.000} C_DIS
LIN {X -134.670,Y 157.062,Z -64.500,A 0.015,B -0.000,C -180.000} C_DIS
LIN {X -134.949,Y 156.639,Z -64.500,A 0.015,B 0.000,C -180.000} C_DIS
LIN {X -136.369,Y 154.801,Z -64.500,A 0.015,B -0.000,C 180.000} C_DIS
LIN {X -136.616,Y 154.516,Z -64.500,A 0.015,B 0.000,C -180.000} C_DIS
LIN {X -137.731,Y 153.364,Z -64.500,A 0.015,B -0.000,C 180.000} C_DIS
LIN {X -138.024,Y 153.095,Z -64.500,A 0.015,B -0.000,C 180.000} C_DIS
LIN {X -140.926,Y 150.729,Z -64.500,A 0.015,B 0.000,C -180.000} C_DIS
LIN {X -141.160,Y 150.554,Z -64.500,A 0.015,B -0.000,C 180.000} C_DIS
LIN {X -142.611,Y 149.566,Z -64.500,A 0.015,B 0.000,C -180.000} C_DIS
LIN {X -142.821,Y 149.434,Z -64.500,A 0.015,B 0.000,C 180.000} C_DIS
LIN {X -179.100,Y 128.454,Z -64.500,A 0.015,B 0.000,C 180.000} C_DIS
CIRC {X -179.556,Y 128.234,Z -64.500,A 0.015,B 0.000,C 180.000},{X -180.040,Y 128.085,Z -64.500,A 0.015,B -0.000,C 180.000} C_DIS
LIN {X -181.129,Y 127.836,Z -64.500,A 0.015,B 0.000,C 180.000} C_DIS
CIRC {X -181.663,Y 127.758,Z -64.500,A 0.015,B 0.000,C 180.000},{X -182.204,Y 127.766,Z -64.500,A 0.015,B 0.000,C -180.000} C_DIS
LIN {X -183.292,Y 127.871,Z -64.500,A 0.015,B 0.000,C 180.000} C_DIS
CIRC {X -183.828,Y 127.966,Z -64.500,A 0.015,B 0.000,C 180.000},{X -184.341,Y 128.146,Z -64.500,A 0.015,B 0.000,C 180.000} C_DIS
LIN {X -185.374,Y 128.604,Z -64.500,A 0.015,B -0.000,C -180.000} C_DIS
LIN {X -186.196,Y 129.120,Z -64.500,A 0.015,B 0.000,C -180.000} C_DIS
LIN {X -186.851,Y 129.678,Z -64.500,A 0.015,B 0.000,C -180.000} C_DIS
LIN {X -187.468,Y 130.371,Z -64.500,A 0.015,B -0.000,C 180.000} C_DIS
LIN {X -188.047,Y 131.236,Z -64.500,A 0.015,B 0.000,C 180.000} C_DIS
LIN {X -188.465,Y 132.107,Z -64.500,A 0.015,B 0.000,C -180.000} C_DIS
LIN {X -188.746,Y 133.004,Z -64.500,A 0.015,B 0.000,C 180.000} C_DIS
CIRC {X -188.862,Y 133.505,Z -64.500,A 0.015,B 0.000,C 180.000},{X -188.901,Y 134.017,Z -64.500,A 0.015,B 0.000,C -180.000} C_DIS
LIN {X -188.846,Y 267.359,Z -64.500,A 0.015,B -0.000,C -180.000} C_DIS
LIN {X -204.666,Y 267.359,Z -64.500,A 0.015,B 0.000,C 180.000} C_DIS
LIN {X -204.611,Y 134.017,Z -64.500,A 0.015,B 0.000,C -180.000} C_DIS
CIRC {X -204.650,Y 133.505,Z -64.500,A 0.015,B 0.000,C 180.000},{X -204.766,Y 133.004,Z -64.500,A 0.015,B -0.000,C 180.000} C_DIS
LIN {X -205.047,Y 132.107,Z -64.500,A 0.015,B 0.000,C -180.000} C_DIS
LIN {X -205.464,Y 131.236,Z -64.500,A 0.015,B 0.000,C -180.000} C_DIS
LIN {X -206.044,Y 130.371,Z -64.500,A 0.015,B 0.000,C -180.000} C_DIS
LIN {X -206.661,Y 129.678,Z -64.500,A 0.015,B 0.000,C -180.000} C_DIS
LIN {X -207.316,Y 129.120,Z -64.500,A 0.015,B 0.000,C -180.000} C_DIS
LIN {X -208.138,Y 128.604,Z -64.500,A 0.015,B 0.000,C -180.000} C_DIS
LIN {X -209.171,Y 128.146,Z -64.500,A 0.015,B 0.000,C -180.000} C_DIS
CIRC {X -209.684,Y 127.966,Z -64.500,A 0.015,B 0.000,C -180.000},{X -210.220,Y 127.871,Z -64.500,A 0.015,B 0.000,C -180.000} C_DIS
LIN {X -211.308,Y 127.766,Z -64.500,A 0.015,B 0.000,C 180.000} C_DIS
CIRC {X -211.849,Y 127.758,Z -64.500,A 0.015,B 0.000,C 180.000},{X -212.383,Y 127.836,Z -64.500,A 0.015,B 0.000,C 180.000} C_DIS
LIN {X -213.472,Y 128.085,Z -64.500,A 0.015,B 0.000,C -180.000} C_DIS
CIRC {X -213.956,Y 128.234,Z -64.500,A 0.015,B -0.000,C 180.000},{X -214.412,Y 128.454,Z -64.500,A 0.015,B 0.000,C 180.000} C_DIS
LIN {X -250.691,Y 149.434,Z -64.500,A 0.015,B 0.000,C 180.000} C_DIS
LIN {X -250.945,Y 149.597,Z -64.500,A 0.015,B 0.000,C 180.000} C_DIS
LIN {X -253.223,Y 151.202,Z -64.500,A 0.015,B 0.000,C -180.000} C_DIS
LIN {X -253.455,Y 151.381,Z -64.500,A 0.015,B 0.000,C -180.000} C_DIS
LIN {X -255.531,Y 153.131,Z -64.500,A 0.015,B -0.000,C -180.000} C_DIS
LIN {X -255.842,Y 153.428,Z -64.500,A 0.015,B 0.000,C -180.000} C_DIS
LIN {X -257.463,Y 155.193,Z -64.500,A 0.015,B 0.000,C -180.000} C_DIS
LIN {X -257.747,Y 155.547,Z -64.500,A 0.015,B -0.000,C -180.000} C_DIS
LIN {X -259.028,Y 157.385,Z -64.500,A 0.015,B 0.000,C -180.000} C_DIS
LIN {X -259.328,Y 157.910,Z -64.500,A 0.015,B -0.000,C 180.000} C_DIS
LIN {X -259.867,Y 159.087,Z -64.500,A 0.015,B -0.000,C 180.000} C_DIS
LIN {X -260.033,Y 159.526,Z -64.500,A 0.015,B -0.000,C -180.000} C_DIS
LIN {X -260.358,Y 160.615,Z -64.500,A 0.015,B 0.000,C 180.000} C_DIS
LIN {X -260.491,Y 161.326,Z -64.500,A 0.015,B 0.000,C 180.000} C_DIS
LIN {X -260.658,Y 163.502,Z -64.500,A 0.015,B 0.000,C -180.000} C_DIS
LIN {X -260.651,Y 164.098,Z -64.500,A 0.015,B 0.000,C 180.000} C_DIS
LIN {X -247.102,Y 299.403,Z -64.500,A 0.015,B 0.000,C 180.000} C_DIS
LIN {X -247.085,Y 299.539,Z -64.500,A 0.015,B 0.000,C -180.000} C_DIS
LIN {X -246.675,Y 302.441,Z -64.500,A 0.015,B -0.000,C 180.000} C_DIS
LIN {X -246.628,Y 302.701,Z -64.500,A 0.015,B 0.000,C -180.000} C_DIS
LIN {X -245.983,Y 305.603,Z -64.500,A 0.015,B -0.000,C 180.000} C_DIS
LIN {X -245.925,Y 305.828,Z -64.500,A 0.015,B -0.000,C 180.000} C_DIS
LIN {X -244.985,Y 309.008,Z -64.500,A 0.015,B 0.000,C 180.000} C_DIS
LIN {X -244.911,Y 309.230,Z -64.500,A 0.015,B 0.000,C 180.000} C_DIS
LIN {X -243.800,Y 312.216,Z -64.500,A 0.015,B 0.000,C -180.000} C_DIS
LIN {X -243.560,Y 312.725,Z -64.500,A 0.015,B 0.000,C -180.000} C_DIS
LIN {X -238.126,Y 322.156,Z -64.500,A 0.015,B -0.000,C 180.000} C_DIS
LIN {X -237.788,Y 322.640,Z -64.500,A 0.015,B 0.000,C 180.000} C_DIS
LIN {X -236.268,Y 324.454,Z -64.500,A 0.015,B 0.000,C 180.000} C_DIS
LIN {X -235.976,Y 324.761,Z -64.500,A 0.015,B 0.000,C 180.000} C_DIS
LIN {X -228.079,Y 332.086,Z -64.500,A 0.015,B 0.000,C -180.000} C_DIS
LIN {X -227.653,Y 332.422,Z -64.500,A 0.015,B 0.000,C -180.000} C_DIS
LIN {X -226.202,Y 333.388,Z -64.500,A 0.015,B -0.000,C 180.000} C_DIS
LIN {X -225.788,Y 333.623,Z -64.500,A 0.015,B 0.000,C -180.000} C_DIS
LIN {X -215.267,Y 338.657,Z -64.500,A 0.015,B 0.000,C -180.000} C_DIS
LIN {X -214.718,Y 338.864,Z -64.500,A 0.015,B 0.000,C 180.000} C_DIS
LIN {X -213.630,Y 339.168,Z -64.500,A 0.015,B 0.000,C 180.000} C_DIS
LIN {X -213.493,Y 339.203,Z -64.500,A 0.015,B 0.000,C -180.000} C_DIS
LIN {X -398.924,Y 339.199,Z -64.500,A 0.015,B -0.000,C -180.000} C_DIS
LIN {X -400.134,Y 339.006,Z -64.500,A 0.015,B 0.000,C -180.000} C_DIS
LIN {X -400.596,Y 338.832,Z -64.500,A 0.015,B 0.000,C -180.000} C_DIS
LIN {X -401.110,Y 338.472,Z -64.330,A 0.015,B 0.000,C -180.000} C_DIS
LIN {X -401.343,Y 338.072,Z -63.865,A 0.015,B 0.000,C 180.000} C_DIS
LIN {X -401.390,Y 337.909,Z -63.230,A 0.015,B 0.000,C 180.000} C_DIS
$VEL.CP = 1.00000
LIN {X -401.390,Y 337.909,Z 11.769,A 0.015,B 0.000,C 180.000} C_DIS
$VEL.CP = 1.00000
LIN {X 5.555,Y -23.879,Z 11.769,A 0.015,B 0.000,C 180.000} C_DIS
$VEL.CP = 0.10000
LIN {X 5.573,Y -23.718,Z 11.147,A 0.015,B -0.000,C 180.000} C_DIS
LIN {X 5.601,Y -23.272,Z 10.684,A 0.015,B 0.000,C 180.000} C_DIS
LIN {X 5.586,Y -22.656,Z 10.500,A 0.015,B 0.000,C 180.000} C_DIS
LIN {X 1.562,Y -17.420,Z 10.256,A 0.015,B -0.000,C -180.000} C_DIS
LIN {X -4.849,Y -19.008,Z 10.012,A 0.015,B -0.000,C 180.000} C_DIS
LIN {X -5.962,Y -25.518,Z 9.768,A 0.015,B 0.000,C 180.000} C_DIS
LIN {X -0.444,Y -29.147,Z 9.524,A 0.015,B 0.000,C -180.000} C_DIS
LIN {X 5.092,Y -25.545,Z 9.280,A 0.015,B -0.000,C 180.000} C_DIS
LIN {X 4.010,Y -19.030,Z 9.036,A 0.015,B 0.000,C -180.000} C_DIS
LIN {X -2.392,Y -17.410,Z 8.792,A 0.015,B 0.000,C -180.000} C_DIS
LIN {X -6.442,Y -22.627,Z 8.548,A 0.015,B 0.000,C -180.000} C_DIS
LIN {X -3.285,Y -28.428,Z 8.304,A 0.015,B 0.000,C -180.000} C_DIS
LIN {X 3.295,Y -27.860,Z 8.060,A 0.015,B 0.000,C 180.000} C_DIS
LIN {X 5.411,Y -21.604,Z 7.815,A 0.015,B 0.000,C 180.000} C_DIS
LIN {X 0.528,Y -17.158,Z 7.571,A 0.015,B 0.000,C -180.000} C_DIS
LIN {X -5.503,Y -19.851,Z 7.327,A 0.015,B 0.000,C -180.000} C_DIS
LIN {X -5.452,Y -26.455,Z 7.083,A 0.015,B 0.000,C -180.000} C_DIS
LIN {X 0.619,Y -29.055,Z 6.839,A 0.015,B 0.000,C 180.000} C_DIS
LIN {X 5.434,Y -24.534,Z 6.595,A 0.015,B 0.000,C -180.000} C_DIS
LIN {X 3.222,Y -18.312,Z 6.351,A 0.015,B 0.000,C -180.000} C_DIS
LIN {X -3.366,Y -17.845,Z 6.107,A 0.015,B 0.000,C -180.000} C_DIS
LIN {X -6.434,Y -23.694,Z 5.863,A 0.015,B 0.000,C -180.000} C_DIS
LIN {X -2.304,Y -28.848,Z 5.619,A 0.015,B 0.000,C 180.000} C_DIS
LIN {X 4.073,Y -27.130,Z 5.375,A 0.015,B 0.000,C 180.000} C_DIS
LIN {X 5.054,Y -20.599,Z 5.131,A 0.015,B -0.000,C 180.000} C_DIS
LIN {X -0.536,Y -17.083,Z 4.887,A 0.015,B 0.000,C 180.000} C_DIS
LIN {X -5.998,Y -20.795,Z 4.643,A 0.015,B 0.000,C 180.000} C_DIS
LIN {X -4.785,Y -27.287,Z 4.399,A 0.015,B 0.000,C 180.000} C_DIS
LIN {X 1.649,Y -28.777,Z 4.155,A 0.015,B 0.000,C 180.000} C_DIS
LIN {X 5.592,Y -23.480,Z 3.911,A 0.015,B -0.000,C -180.000} C_DIS
LIN {X 2.319,Y -17.744,Z 3.667,A 0.015,B 0.000,C 180.000} C_DIS
LIN {X -4.248,Y -18.445,Z 3.423,A 0.015,B 0.000,C 180.000} C_DIS
LIN {X -6.238,Y -24.742,Z 3.179,A 0.015,B -0.000,C 180.000} C_DIS
LIN {X -1.265,Y -29.088,Z 2.935,A 0.015,B 0.000,C 180.000} C_DIS
LIN {X 4.710,Y -26.274,Z 2.690,A 0.015,B 0.000,C -180.000} C_DIS
LIN {X 4.525,Y -19.672,Z 2.446,A 0.015,B 0.000,C -180.000} C_DIS
LIN {X -1.597,Y -17.196,Z 2.202,A 0.015,B 0.000,C 180.000} C_DIS
LIN {X -6.319,Y -21.813,Z 1.958,A 0.015,B 0.000,C -180.000} C_DIS
LIN {X -3.982,Y -27.989,Z 1.714,A 0.015,B -0.000,C -180.000} C_DIS
LIN {X 2.614,Y -28.323,Z 1.470,A 0.015,B -0.000,C 180.000} C_DIS
LIN {X 5.563,Y -22.413,Z 1.226,A 0.015,B -0.000,C -180.000} C_DIS
LIN {X 1.330,Y -17.344,Z 0.982,A 0.015,B 0.000,C -180.000} C_DIS
LIN {X -5.011,Y -19.190,Z 0.738,A 0.015,B 0.000,C 180.000} C_DIS
LIN {X -5.860,Y -25.740,Z 0.494,A 0.015,B 0.000,C 180.000} C_DIS
LIN {X -0.200,Y -29.142,Z 0.250,A 0.015,B 0.000,C 180.000} C_DIS
LIN {X 5.186,Y -25.320,Z 0.006,A 0.015,B -0.000,C -180.000} C_DIS
LIN {X 3.842,Y -18.854,Z -0.238,A 0.015,B 0.000,C 180.000} C_DIS
LIN {X -2.621,Y -17.494,Z -0.482,A 0.015,B 0.000,C -180.000} C_DIS
LIN {X -6.457,Y -22.870,Z -0.726,A 0.015,B 0.000,C -180.000} C_DIS
LIN {X -3.068,Y -28.539,Z -0.970,A 0.015,B 0.000,C 180.000} C_DIS
LIN {X 3.484,Y -27.705,Z -1.214,A 0.015,B 0.000,C 180.000} C_DIS
LIN {X 5.346,Y -21.369,Z -1.458,A 0.015,B 0.000,C 180.000} C_DIS
LIN {X 0.286,Y -17.124,Z -1.702,A 0.015,B 0.000,C 180.000} C_DIS
LIN {X -5.630,Y -20.059,Z -1.946,A 0.015,B 0.000,C -180.000} C_DIS
LIN {X -5.313,Y -26.655,Z -2.190,A 0.015,B 0.000,C 180.000} C_DIS
LIN {X 0.858,Y -29.008,Z -2.435,A 0.015,B 0.000,C 180.000} C_DIS
LIN {X 5.486,Y -24.296,Z -2.679,A 0.015,B -0.000,C 180.000} C_DIS
LIN {X 3.025,Y -18.168,Z -2.923,A 0.015,B 0.000,C 180.000} C_DIS
LIN {X -3.577,Y -17.968,Z -3.167,A 0.015,B 0.000,C 180.000} C_DIS
LIN {X -6.405,Y -23.936,Z -3.411,A 0.015,B 0.000,C 180.000} C_DIS
LIN {X -2.071,Y -28.919,Z -3.655,A 0.015,B 0.000,C -180.000} C_DIS
LIN {X 4.231,Y -26.945,Z -3.899,A 0.015,B 0.000,C 180.000} C_DIS
LIN {X 4.948,Y -20.379,Z -4.143,A 0.015,B -0.000,C 180.000} C_DIS
LIN {X -0.780,Y -17.092,Z -4.387,A 0.015,B 0.000,C -180.000} C_DIS
LIN {X -6.087,Y -21.022,Z -4.631,A 0.015,B 0.000,C 180.000} C_DIS
LIN {X -4.613,Y -27.460,Z -4.875,A 0.015,B 0.000,C 180.000} C_DIS
LIN {X 1.876,Y -28.689,Z -5.119,A 0.015,B 0.000,C -180.000} C_DIS
LIN {X 5.602,Y -23.236,Z -5.363,A 0.015,B 0.000,C -180.000} C_DIS
LIN {X 2.099,Y -17.637,Z -5.607,A 0.015,B 0.000,C 180.000} C_DIS
LIN {X -4.434,Y -18.603,Z -5.851,A 0.015,B 0.000,C 180.000} C_DIS
LIN {X -6.167,Y -24.976,Z -6.095,A 0.015,B -0.000,C -180.000} C_DIS
LIN {X -1.023,Y -29.117,Z -6.339,A 0.015,B 0.000,C -180.000} C_DIS
LIN {X 4.833,Y -26.064,Z -6.583,A 0.015,B 0.000,C 180.000} C_DIS
LIN {X 4.382,Y -19.475,Z -6.827,A 0.015,B 0.000,C -180.000} C_DIS
LIN {X -1.835,Y -17.248,Z -7.071,A 0.015,B 0.000,C -180.000} C_DIS
LIN {X -6.367,Y -22.052,Z -7.315,A 0.015,B -0.000,C 180.000} C_DIS
LIN {X -3.782,Y -28.129,Z -7.560,A 0.015,B 0.000,C 180.000} C_DIS
LIN {X 2.822,Y -28.196,Z -7.804,A 0.015,B 0.000,C 180.000} C_DIS
LIN {X 5.529,Y -22.172,Z -8.048,A 0.015,B 0.000,C 180.000} C_DIS
LIN {X 1.095,Y -17.277,Z -8.292,A 0.015,B 0.000,C 180.000} C_DIS
LIN {X -5.166,Y -19.379,Z -8.536,A 0.015,B 0.000,C 180.000} C_DIS
LIN {X -5.750,Y -25.957,Z -8.780,A 0.015,B 0.000,C 180.000} C_DIS
LIN {X 0.044,Y -29.128,Z -9.024,A 0.015,B 0.000,C -180.000} C_DIS
LIN {X 5.270,Y -25.091,Z -9.268,A 0.015,B 0.000,C 180.000} C_DIS
LIN {X 3.666,Y -18.684,Z -9.512,A 0.015,B 0.000,C 180.000} C_DIS
LIN {X -2.847,Y -17.587,Z -9.756,A 0.015,B 0.000,C -180.000} C_DIS
LIN {X -6.462,Y -23.114,Z -10.000,A 0.015,B -0.000,C -180.000} C_DIS
CIRC {X -4.819,Y -27.079,Z -10.000,A 0.015,B -0.000,C 180.000},{X -0.854,Y -28.721,Z -10.000,A 0.015,B 0.000,C -180.000} C_DIS
CIRC {X 3.111,Y -27.079,Z -10.000,A 0.015,B 0.000,C 180.000},{X 4.753,Y -23.114,Z -10.000,A 0.015,B 0.000,C -180.000} C_DIS
LIN {X 4.753,Y -20.363,Z -10.000,A 0.015,B 0.000,C 180.000} C_DIS
CIRC {X 3.647,Y -18.799,Z -10.000,A 0.015,B 0.000,C -180.000},{X 1.804,Y -19.321,Z -10.000,A 0.015,B 0.000,C -180.000} C_DIS
LIN {X -0.810,Y -22.561,Z -10.000,A 0.015,B 0.000,C 180.000} C_DIS
CIRC {X -1.052,Y -24.632,Z -10.000,A 0.015,B 0.000,C -180.000},{X 0.711,Y -25.744,Z -10.000,A 0.015,B 0.000,C -180.000} C_DIS
LIN {X 2.639,Y -25.744,Z -10.000,A 0.015,B 0.000,C 180.000} C_DIS
CIRC {X 4.134,Y -25.125,Z -10.000,A 0.015,B 0.000,C -180.000},{X 4.753,Y -23.630,Z -10.000,A 0.015,B 0.000,C 180.000} C_DIS
LIN {X 4.753,Y -23.114,Z -10.000,A 0.015,B 0.000,C -180.000} C_DIS
LIN {X 3.541,Y -23.379,Z -10.000,A 0.015,B 0.000,C 180.000} C_DIS
LIN {X 4.031,Y -24.448,Z -10.000,A 0.015,B 0.000,C 180.000} C_DIS
LIN {X 4.228,Y -24.691,Z -10.000,A 0.015,B -0.000,C 180.000} C_DIS
LIN {X 8.680,Y -28.027,Z -10.000,A 0.015,B 0.000,C -180.000} C_DIS
LIN {X 9.366,Y -28.668,Z -10.000,A 0.015,B 0.000,C 180.000} C_DIS
LIN {X 9.675,Y -28.604,Z -10.000,A 0.015,B 0.000,C 180.000} C_DIS
LIN {X 10.021,Y -27.803,Z -10.000,A 0.015,B 0.000,C 180.000} C_DIS
LIN {X 10.218,Y -26.938,Z -10.000,A 0.015,B 0.000,C -180.000} C_DIS
LIN {X 10.275,Y -25.867,Z -10.000,A 0.015,B 0.000,C -180.000} C_DIS
LIN {X 10.274,Y 7.531,Z -10.000,A 0.015,B 0.000,C -180.000} C_DIS
LIN {X 6.199,Y -2.885,Z -10.000,A 0.015,B 0.000,C 180.000} C_DIS
LIN {X 5.976,Y -3.347,Z -10.000,A 0.015,B 0.000,C -180.000} C_DIS
LIN {X 1.986,Y -10.239,Z -10.000,A 0.015,B 0.000,C -180.000} C_DIS
LIN {X 1.691,Y -10.668,Z -10.000,A 0.015,B 0.000,C -180.000} C_DIS
LIN {X -6.460,Y -20.770,Z -10.000,A 0.015,B 0.000,C 180.000} C_DIS
LIN {X -7.171,Y -21.429,Z -10.000,A 0.015,B 0.000,C -180.000} C_DIS
LIN {X -10.538,Y -23.754,Z -10.000,A 0.015,B 0.000,C -180.000} C_DIS
LIN {X -10.599,Y -23.795,Z -10.000,A 0.015,B -0.000,C 180.000} C_DIS
LIN {X -18.171,Y -28.781,Z -10.000,A 0.015,B 0.000,C 180.000} C_DIS
LIN {X -18.860,Y -29.129,Z -10.000,A 0.015,B 0.000,C -180.000} C_DIS
LIN {X -19.996,Y -29.548,Z -10.000,A 0.015,B 0.000,C -180.000} C_DIS
LIN {X -20.242,Y -29.628,Z -10.000,A 0.015,B 0.000,C -180.000} C_DIS
LIN {X -26.002,Y -31.266,Z -10.000,A 0.015,B 0.000,C -180.000} C_DIS
LIN {X 5.412,Y -31.266,Z -10.000,A 0.015,B 0.000,C 180.000} C_DIS
LIN {X 6.622,Y -31.073,Z -10.000,A 0.015,B 0.000,C -180.000} C_DIS
$VEL.CP = 1.00000
LIN {X 6.622,Y -31.073,Z 11.000,A 0.015,B 0.000,C 180.000} C_DIS
$VEL.CP = 1.00000
LIN {X 5.565,Y -23.893,Z 11.000,A 0.015,B 0.000,C -180.000} C_DIS
$VEL.CP = 1.00000
LIN {X 5.565,Y -23.893,Z 1.769,A 0.015,B 0.000,C 180.000} C_DIS
$VEL.CP = 0.10000
LIN {X 5.584,Y -23.731,Z 1.147,A 0.015,B 0.000,C 180.000} C_DIS
LIN {X 5.612,Y -23.286,Z 0.684,A 0.015,B 0.000,C -180.000} C_DIS
LIN {X 5.596,Y -22.670,Z 0.500,A 0.015,B 0.000,C 180.000} C_DIS
LIN {X 1.572,Y -17.433,Z 0.256,A 0.015,B 0.000,C -180.000} C_DIS
LIN {X -4.838,Y -19.022,Z 0.012,A 0.015,B -0.000,C 180.000} C_DIS
LIN {X -5.952,Y -25.532,Z -0.232,A 0.015,B -0.000,C 180.000} C_DIS
LIN {X -0.433,Y -29.160,Z -0.476,A 0.015,B 0.000,C -180.000} C_DIS
LIN {X 5.102,Y -25.559,Z -0.720,A 0.015,B 0.000,C -180.000} C_DIS
LIN {X 4.021,Y -19.044,Z -0.964,A 0.015,B 0.000,C 180.000} C_DIS
LIN {X -2.382,Y -17.424,Z -1.208,A 0.015,B 0.000,C 180.000} C_DIS
LIN {X -6.431,Y -22.641,Z -1.452,A 0.015,B 0.000,C 180.000} C_DIS
LIN {X -3.275,Y -28.442,Z -1.696,A 0.015,B 0.000,C -180.000} C_DIS
LIN {X 3.305,Y -27.874,Z -1.940,A 0.015,B 0.000,C -180.000} C_DIS
LIN {X 5.422,Y -21.618,Z -2.185,A 0.015,B 0.000,C -180.000} C_DIS
LIN {X 0.538,Y -17.172,Z -2.429,A 0.015,B 0.000,C 180.000} C_DIS
LIN {X -5.492,Y -19.865,Z -2.673,A 0.015,B -0.000,C -180.000} C_DIS
LIN {X -5.442,Y -26.469,Z -2.917,A 0.015,B 0.000,C 180.000} C_DIS
LIN {X 0.629,Y -29.069,Z -3.161,A 0.015,B 0.000,C -180.000} C_DIS
LIN {X 5.444,Y -24.548,Z -3.405,A 0.015,B 0.000,C 180.000} C_DIS
LIN {X 3.232,Y -18.325,Z -3.649,A 0.015,B 0.000,C 180.000} C_DIS
LIN {X -3.356,Y -17.859,Z -3.893,A 0.015,B 0.000,C -180.000} C_DIS
LIN {X -6.423,Y -23.707,Z -4.137,A 0.015,B 0.000,C 180.000} C_DIS
LIN {X -2.294,Y -28.862,Z -4.381,A 0.015,B 0.000,C 180.000} C_DIS
LIN {X 4.083,Y -27.144,Z -4.625,A 0.015,B 0.000,C 180.000} C_DIS
LIN {X 5.064,Y -20.613,Z -4.869,A 0.015,B 0.000,C 180.000} C_DIS
LIN {X -0.526,Y -17.096,Z -5.113,A 0.015,B 0.000,C -180.000} C_DIS
LIN {X -5.988,Y -20.809,Z -5.357,A 0.015,B -0.000,C 180.000} C_DIS
LIN {X -4.775,Y -27.301,Z -5.601,A 0.015,B 0.000,C -180.000} C_DIS
LIN {X 1.659,Y -28.791,Z -5.845,A 0.015,B 0.000,C -180.000} C_DIS
LIN {X 5.603,Y -23.493,Z -6.089,A 0.015,B 0.000,C 180.000} C_DIS
LIN {X 2.329,Y -17.758,Z -6.333,A 0.015,B 0.000,C -180.000} C_DIS
LIN {X -4.238,Y -18.458,Z -6.577,A 0.015,B 0.000,C -180.000} C_DIS
LIN {X -6.227,Y -24.756,Z -6.821,A 0.015,B -0.000,C -180.000} C_DIS
LIN {X -1.255,Y -29.102,Z -7.065,A 0.015,B -0.000,C 180.000} C_DIS
LIN {X 4.720,Y -26.288,Z -7.310,A 0.015,B 0.000,C 180.000} C_DIS
LIN {X 4.536,Y -19.686,Z -7.554,A 0.015,B -0.000,C -180.000} C_DIS
LIN {X -1.587,Y -17.210,Z -7.798,A 0.015,B 0.000,C 180.000} C_DIS
LIN {X -6.309,Y -21.826,Z -8.042,A 0.015,B -0.000,C 180.000} C_DIS
LIN {X -3.972,Y -28.003,Z -8.286,A 0.015,B 0.000,C 180.000} C_DIS
LIN {X 2.624,Y -28.337,Z -8.530,A 0.015,B 0.000,C 180.000} C_DIS
LIN {X 5.573,Y -22.427,Z -8.774,A 0.015,B 0.000,C 180.000} C_DIS
LIN {X 1.340,Y -17.358,Z -9.018,A 0.015,B 0.000,C 180.000} C_DIS
LIN {X -5.001,Y -19.204,Z -9.262,A 0.015,B -0.000,C -180.000} C_DIS
LIN {X -5.850,Y -25.753,Z -9.506,A 0.015,B 0.000,C -180.000} C_DIS
LIN {X -0.189,Y -29.156,Z -9.750,A 0.015,B -0.000,C 180.000} C_DIS
LIN {X 5.196,Y -25.333,Z -9.994,A 0.015,B 0.000,C 180.000} C_DIS
LIN {X 3.852,Y -18.867,Z -10.238,A 0.015,B 0.000,C 180.000} C_DIS
LIN {X -2.611,Y -17.508,Z -10.482,A 0.015,B 0.000,C 180.000} C_DIS
LIN {X -6.446,Y -22.884,Z -10.726,A 0.015,B -0.000,C 180.000} C_DIS
LIN {X -3.057,Y -28.553,Z -10.970,A 0.015,B 0.000,C 180.000} C_DIS
LIN {X 3.494,Y -27.719,Z -11.214,A 0.015,B 0.000,C -180.000} C_DIS
LIN {X 5.356,Y -21.383,Z -11.458,A 0.015,B 0.000,C 180.000} C_DIS
LIN {X 0.296,Y -17.138,Z -11.702,A 0.015,B 0.000,C 180.000} C_DIS
LIN {X -5.620,Y -20.072,Z -11.946,A 0.015,B 0.000,C -180.000} C_DIS
LIN {X -5.302,Y -26.669,Z -12.190,A 0.015,B 0.000,C -180.000} C_DIS
LIN {X 0.869,Y -29.021,Z -12.435,A 0.015,B -0.000,C -180.000} C_DIS
LIN {X 5.497,Y -24.310,Z -12.679,A 0.015,B 0.000,C -180.000} C_DIS
LIN {X 3.035,Y -18.182,Z -12.923,A 0.015,B 0.000,C 180.000} C_DIS
LIN {X -3.566,Y -17.982,Z -13.167,A 0.015,B 0.000,C -180.000} C_DIS
LIN {X -6.395,Y -23.950,Z -13.411,A 0.015,B 0.000,C 180.000} C_DIS
LIN {X -2.061,Y -28.933,Z -13.655,A 0.015,B 0.000,C 180.000} C_DIS
LIN {X 4.242,Y -26.958,Z -13.899,A 0.015,B 0.000,C -180.000} C_DIS
LIN {X 4.958,Y -20.393,Z -14.143,A 0.015,B 0.000,C -180.000} C_DIS
LIN {X -0.770,Y -17.106,Z -14.387,A 0.015,B 0.000,C -180.000} C_DIS
LIN {X -6.077,Y -21.036,Z -14.631,A 0.015,B 0.000,C -180.000} C_DIS
LIN {X -4.602,Y -27.474,Z -14.875,A 0.015,B -0.000,C 180.000} C_DIS
LIN {X 1.887,Y -28.703,Z -15.119,A 0.015,B 0.000,C 180.000} C_DIS
LIN {X 5.613,Y -23.250,Z -15.363,A 0.015,B 0.000,C 180.000} C_DIS
LIN {X 2.110,Y -17.651,Z -15.607,A 0.015,B 0.000,C -180.000} C_DIS
LIN {X -4.424,Y -18.617,Z -15.851,A 0.015,B -0.000,C 180.000} C_DIS
LIN {X -6.157,Y -24.989,Z -16.095,A 0.015,B 0.000,C 180.000} C_DIS
LIN {X -1.013,Y -29.131,Z -16.339,A 0.015,B 0.000,C 180.000} C_DIS
LIN {X 4.843,Y -26.078,Z -16.583,A 0.015,B 0.000,C 180.000} C_DIS
LIN {X 4.393,Y -19.489,Z -16.827,A 0.015,B 0.000,C -180.000} C_DIS
LIN {X -1.825,Y -17.262,Z -17.071,A 0.015,B 0.000,C -180.000} C_DIS
LIN {X -6.357,Y -22.066,Z -17.315,A 0.015,B -0.000,C -180.000} C_DIS
LIN {X -3.772,Y -28.143,Z -17.560,A 0.015,B 0.000,C -180.000} C_DIS
LIN {X 2.832,Y -28.209,Z -17.804,A 0.015,B 0.000,C 180.000} C_DIS
LIN {X 5.540,Y -22.185,Z -18.048,A 0.015,B 0.000,C 180.000} C_DIS
LIN {X 1.106,Y -17.291,Z -18.292,A 0.015,B 0.000,C -180.000} C_DIS
LIN {X -5.156,Y -19.392,Z -18.536,A 0.015,B 0.000,C -180.000} C_DIS
LIN {X -5.739,Y -25.971,Z -18.780,A 0.015,B 0.000,C 180.000} C_DIS
LIN {X 0.054,Y -29.142,Z -19.024,A 0.015,B 0.000,C 180.000} C_DIS
LIN {X 5.281,Y -25.105,Z -19.268,A 0.015,B 0.000,C 180.000} C_DIS
LIN {X 3.676,Y -18.698,Z -19.512,A 0.015,B 0.000,C 180.000} C_DIS
LIN {X -2.836,Y -17.601,Z -19.756,A 0.015,B -0.000,C 180.000} C_DIS
LIN {X -6.451,Y -23.128,Z -20.000,A 0.015,B 0.000,C -180.000} C_DIS
CIRC {X -4.809,Y -27.092,Z -20.000,A 0.015,B 0.000,C 180.000},{X -0.844,Y -28.734,Z -20.000,A 0.015,B 0.000,C 180.000} C_DIS
CIRC {X 3.120,Y -27.092,Z -20.000,A 0.015,B 0.000,C 180.000},{X 4.762,Y -23.128,Z -20.000,A 0.015,B 0.000,C 180.000} C_DIS
LIN {X 4.762,Y -20.362,Z -20.000,A 0.015,B 0.000,C 180.000} C_DIS
CIRC {X 3.656,Y -18.801,Z -20.000,A 0.015,B 0.000,C 180.000},{X 1.817,Y -19.328,Z -20.000,A 0.015,B 0.000,C -180.000} C_DIS
LIN {X -0.777,Y -22.567,Z -20.000,A 0.015,B -0.000,C -180.000} C_DIS
CIRC {X -1.015,Y -24.641,Z -20.000,A 0.015,B -0.000,C -180.000},{X 0.753,Y -25.753,Z -20.000,A 0.015,B 0.000,C 180.000} C_DIS
LIN {X 2.648,Y -25.753,Z -20.000,A 0.015,B 0.000,C -180.000} C_DIS
CIRC {X 4.143,Y -25.134,Z -20.000,A 0.015,B 0.000,C -180.000},{X 4.762,Y -23.639,Z -20.000,A 0.015,B 0.000,C -180.000} C_DIS
LIN {X 4.762,Y -23.128,Z -20.000,A 0.015,B 0.000,C -180.000} C_DIS
LIN {X 3.550,Y -23.394,Z -20.000,A 0.015,B 0.000,C 180.000} C_DIS
LIN {X 4.042,Y -24.459,Z -20.000,A 0.015,B 0.000,C 180.000} C_DIS
LIN {X 4.238,Y -24.701,Z -20.000,A 0.015,B 0.000,C -180.000} C_DIS
LIN {X 8.680,Y -28.027,Z -20.000,A 0.015,B -0.000,C 180.000} C_DIS
LIN {X 9.366,Y -28.668,Z -20.000,A 0.015,B 0.000,C 180.000} C_DIS
LIN {X 9.675,Y -28.604,Z -20.000,A 0.015,B 0.000,C -180.000} C_DIS
LIN {X 10.021,Y -27.803,Z -20.000,A 0.015,B 0.000,C 180.000} C_DIS
LIN {X 10.218,Y -26.938,Z -20.000,A 0.015,B -0.000,C -180.000} C_DIS
LIN {X 10.275,Y -25.867,Z -20.000,A 0.015,B -0.000,C -180.000} C_DIS
LIN {X 10.274,Y 7.501,Z -20.000,A 0.015,B 0.000,C -180.000} C_DIS
LIN {X 6.197,Y -2.888,Z -20.000,A 0.015,B 0.000,C -180.000} C_DIS
LIN {X 5.976,Y -3.347,Z -20.000,A 0.015,B 0.000,C -180.000} C_DIS
LIN {X 1.986,Y -10.239,Z -20.000,A 0.015,B 0.000,C 180.000} C_DIS
LIN {X 1.699,Y -10.659,Z -20.000,A 0.015,B 0.000,C -180.000} C_DIS
LIN {X -6.187,Y -20.501,Z -20.000,A 0.015,B -0.000,C 180.000} C_DIS
LIN {X -6.615,Y -20.946,Z -20.000,A 0.015,B 0.000,C -180.000} C_DIS
LIN {X -7.346,Y -21.577,Z -20.000,A 0.015,B 0.000,C -180.000} C_DIS
LIN {X -7.682,Y -21.833,Z -20.000,A 0.015,B 0.000,C 180.000} C_DIS
LIN {X -17.934,Y -28.664,Z -20.000,A 0.015,B 0.000,C 180.000} C_DIS
LIN {X -18.587,Y -29.002,Z -20.000,A 0.015,B 0.000,C 180.000} C_DIS
LIN {X -19.943,Y -29.528,Z -20.000,A 0.015,B 0.000,C 180.000} C_DIS
LIN {X -20.228,Y -29.625,Z -20.000,A 0.015,B -0.000,C -180.000} C_DIS
LIN {X -25.914,Y -31.266,Z -20.000,A 0.015,B 0.000,C 180.000} C_DIS
LIN {X 5.412,Y -31.266,Z -20.000,A 0.015,B 0.000,C 180.000} C_DIS
LIN {X 6.622,Y -31.073,Z -20.000,A 0.015,B 0.000,C 180.000} C_DIS
LIN {X 7.443,Y -30.763,Z -20.000,A 0.015,B 0.000,C -180.000} C_DIS
LIN {X 7.663,Y -30.627,Z -20.000,A 0.015,B 0.000,C 180.000} C_DIS
LIN {X 7.905,Y -29.139,Z -20.000,A 0.015,B 0.000,C 180.000} C_DIS
LIN {X 5.429,Y -26.154,Z -20.000,A 0.015,B 0.000,C 180.000} C_DIS
LIN {X 5.258,Y -25.176,Z -20.000,A 0.015,B 0.000,C 180.000} C_DIS
LIN {X 3.734,Y -18.753,Z -20.244,A 0.015,B 0.000,C 180.000} C_DIS
LIN {X -2.760,Y -17.571,Z -20.488,A 0.015,B 0.000,C 180.000} C_DIS
LIN {X -6.449,Y -23.044,Z -20.732,A 0.015,B 0.000,C -180.000} C_DIS
LIN {X -2.917,Y -28.620,Z -20.976,A 0.015,B 0.000,C 180.000} C_DIS
LIN {X 3.608,Y -27.623,Z -21.220,A 0.015,B 0.000,C -180.000} C_DIS
LIN {X 5.314,Y -21.246,Z -21.463,A 0.015,B -0.000,C 180.000} C_DIS
LIN {X 0.157,Y -17.125,Z -21.707,A 0.015,B 0.000,C -180.000} C_DIS
LIN {X -5.687,Y -20.193,Z -21.951,A 0.015,B 0.000,C 180.000} C_DIS
LIN {X -5.222,Y -26.778,Z -22.195,A 0.015,B -0.000,C 180.000} C_DIS
LIN {X 0.996,Y -28.995,Z -22.439,A 0.015,B 0.000,C -180.000} C_DIS
LIN {X 5.521,Y -24.189,Z -22.683,A 0.015,B 0.000,C -180.000} C_DIS
LIN {X 2.937,Y -18.116,Z -22.927,A 0.015,B 0.000,C -180.000} C_DIS
LIN {X -3.664,Y -18.045,Z -23.171,A 0.015,B 0.000,C -180.000} C_DIS
LIN {X -6.377,Y -24.063,Z -23.415,A 0.015,B 0.000,C 180.000} C_DIS
LIN {X -1.955,Y -28.963,Z -23.659,A 0.015,B 0.000,C -180.000} C_DIS
LIN {X 4.308,Y -26.879,Z -23.902,A 0.015,B 0.000,C -180.000} C_DIS
LIN {X 4.914,Y -20.306,Z -24.146,A 0.015,B 0.000,C 180.000} C_DIS
LIN {X -0.864,Y -17.114,Z -24.390,A 0.015,B 0.000,C 180.000} C_DIS
LIN {X -6.107,Y -21.124,Z -24.634,A 0.015,B 0.000,C 180.000} C_DIS
LIN {X -4.538,Y -27.536,Z -24.878,A 0.015,B 0.000,C 180.000} C_DIS
LIN {X 1.965,Y -28.672,Z -25.122,A 0.015,B 0.000,C 180.000} C_DIS
LIN {X 5.615,Y -23.173,Z -25.366,A 0.015,B -0.000,C -180.000} C_DIS
LIN {X 2.043,Y -17.622,Z -25.610,A 0.015,B -0.000,C 180.000} C_DIS
LIN {X -4.475,Y -18.666,Z -25.854,A 0.015,B 0.000,C 180.000} C_DIS
LIN {X -6.134,Y -25.054,Z -26.098,A 0.015,B 0.000,C -180.000} C_DIS
LIN {X -0.949,Y -29.139,Z -26.341,A 0.015,B 0.000,C 180.000} C_DIS
LIN {X 4.873,Y -26.029,Z -26.585,A 0.015,B 0.000,C 180.000} C_DIS
LIN {X 4.361,Y -19.448,Z -26.829,A 0.015,B 0.000,C 180.000} C_DIS
LIN {X -1.872,Y -17.275,Z -27.073,A 0.015,B -0.000,C -180.000} C_DIS
LIN {X -6.363,Y -22.113,Z -27.317,A 0.015,B 0.000,C -180.000} C_DIS
LIN {X -3.735,Y -28.168,Z -27.561,A 0.015,B 0.000,C 180.000} C_DIS
LIN {X 2.865,Y -28.191,Z -27.805,A 0.015,B 0.000,C 180.000} C_DIS
LIN {X 5.536,Y -22.155,Z -28.049,A 0.015,B -0.000,C -180.000} C_DIS
LIN {X 1.079,Y -17.286,Z -28.293,A 0.015,B -0.000,C -180.000} C_DIS
LIN {X -5.169,Y -19.414,Z -28.537,A 0.015,B 0.000,C -180.000} C_DIS
LIN {X -5.728,Y -25.991,Z -28.780,A 0.015,B 0.000,C -180.000} C_DIS
LIN {X 0.072,Y -29.142,Z -29.024,A 0.015,B 0.000,C -180.000} C_DIS
LIN {X 5.286,Y -25.095,Z -29.268,A 0.015,B 0.000,C -180.000} C_DIS
LIN {X 3.672,Y -18.695,Z -29.512,A 0.015,B 0.000,C 180.000} C_DIS
LIN {X -2.839,Y -17.605,Z -29.756,A 0.015,B -0.000,C -180.000} C_DIS
LIN {X -6.450,Y -23.130,Z -30.000,A 0.015,B 0.000,C -180.000} C_DIS
CIRC {X -0.843,Y -28.736,Z -30.000,A 0.015,B 0.000,C 180.000},{X 4.763,Y -23.130,Z -30.000,A 0.015,B -0.000,C -180.000} C_DIS
LIN {X 4.763,Y -20.362,Z -30.000,A 0.015,B -0.000,C -180.000} C_DIS
CIRC {X 3.657,Y -18.802,Z -30.000,A 0.015,B 0.000,C -180.000},{X 1.819,Y -19.329,Z -30.000,A 0.015,B -0.000,C -180.000} C_DIS
LIN {X -0.773,Y -22.568,Z -30.000,A 0.015,B 0.000,C 180.000} C_DIS
CIRC {X -1.010,Y -24.642,Z -30.000,A 0.015,B -0.000,C 180.000},{X 0.758,Y -25.754,Z -30.000,A 0.015,B 0.000,C 180.000} C_DIS
LIN {X 2.649,Y -25.754,Z -30.000,A 0.015,B 0.000,C -180.000} C_DIS
CIRC {X 4.144,Y -25.135,Z -30.000,A 0.015,B 0.000,C -180.000},{X 4.763,Y -23.640,Z -30.000,A 0.015,B 0.000,C -180.000} C_DIS
LIN {X 4.763,Y -23.130,Z -30.000,A 0.015,B -0.000,C 180.000} C_DIS
LIN {X 3.552,Y -23.396,Z -30.000,A 0.015,B 0.000,C 180.000} C_DIS
LIN {X 4.044,Y -24.461,Z -30.000,A 0.015,B 0.000,C 180.000} C_DIS
LIN {X 4.240,Y -24.703,Z -30.000,A 0.015,B 0.000,C -180.000} C_DIS
LIN {X 8.680,Y -28.027,Z -30.000,A 0.015,B 0.000,C -180.000} C_DIS
LIN {X 9.366,Y -28.668,Z -30.000,A 0.015,B 0.000,C 180.000} C_DIS
LIN {X 9.675,Y -28.604,Z -30.000,A 0.015,B -0.000,C 180.000} C_DIS
LIN {X 10.021,Y -27.803,Z -30.000,A 0.015,B 0.000,C 180.000} C_DIS
LIN {X 10.218,Y -26.938,Z -30.000,A 0.015,B 0.000,C 180.000} C_DIS
LIN {X 10.275,Y -25.867,Z -30.000,A 0.015,B 0.000,C -180.000} C_DIS
LIN {X 10.274,Y 7.471,Z -30.000,A 0.015,B 0.000,C -180.000} C_DIS
LIN {X 6.196,Y -2.891,Z -30.000,A 0.015,B 0.000,C -180.000} C_DIS
LIN {X 5.976,Y -3.347,Z -30.000,A 0.015,B 0.000,C -180.000} C_DIS
LIN {X 1.986,Y -10.239,Z -30.000,A 0.015,B 0.000,C -180.000} C_DIS
LIN {X 1.700,Y -10.658,Z -30.000,A 0.015,B 0.000,C 180.000} C_DIS
LIN {X -6.175,Y -20.496,Z -30.000,A 0.015,B -0.000,C -180.000} C_DIS
LIN {X -6.615,Y -20.952,Z -30.000,A 0.015,B -0.000,C 180.000} C_DIS
LIN {X -7.357,Y -21.587,Z -30.000,A 0.015,B 0.000,C 180.000} C_DIS
LIN {X -7.675,Y -21.828,Z -30.000,A 0.015,B 0.000,C 180.000} C_DIS
LIN {X -17.706,Y -28.549,Z -30.000,A 0.015,B 0.000,C 180.000} C_DIS
LIN {X -18.187,Y -28.818,Z -30.000,A 0.015,B 0.000,C 180.000} C_DIS
LIN {X -19.197,Y -29.277,Z -30.000,A 0.015,B 0.000,C 180.000} C_DIS
LIN {X -19.641,Y -29.443,Z -30.000,A 0.015,B 0.000,C 180.000} C_DIS
LIN {X -25.814,Y -31.266,Z -30.000,A 0.015,B 0.000,C -180.000} C_DIS
LIN {X 5.412,Y -31.266,Z -30.000,A 0.015,B 0.000,C 180.000} C_DIS
LIN {X 6.622,Y -31.073,Z -30.000,A 0.015,B 0.000,C 180.000} C_DIS
LIN {X 7.443,Y -30.763,Z -30.000,A 0.015,B 0.000,C 180.000} C_DIS
LIN {X 7.663,Y -30.627,Z -30.000,A 0.015,B 0.000,C -180.000} C_DIS
LIN {X 7.905,Y -29.139,Z -30.000,A 0.015,B 0.000,C -180.000} C_DIS
LIN {X 5.430,Y -26.155,Z -30.000,A 0.015,B 0.000,C -180.000} C_DIS
LIN {X 5.259,Y -25.177,Z -30.000,A 0.015,B 0.000,C 180.000} C_DIS
LIN {X 3.736,Y -18.755,Z -30.244,A 0.015,B 0.000,C 180.000} C_DIS
LIN {X -2.759,Y -17.572,Z -30.488,A 0.015,B 0.000,C 180.000} C_DIS
LIN {X -6.448,Y -23.045,Z -30.732,A 0.015,B 0.000,C -180.000} C_DIS
LIN {X -2.916,Y -28.622,Z -30.976,A 0.015,B 0.000,C -180.000} C_DIS
LIN {X 3.609,Y -27.624,Z -31.220,A 0.015,B -0.000,C -180.000} C_DIS
LIN {X 5.315,Y -21.247,Z -31.463,A 0.015,B -0.000,C 180.000} C_DIS
LIN {X 0.158,Y -17.126,Z -31.707,A 0.015,B 0.000,C 180.000} C_DIS
LIN {X -5.686,Y -20.195,Z -31.951,A 0.015,B 0.000,C -180.000} C_DIS
LIN {X -5.221,Y -26.779,Z -32.195,A 0.015,B 0.000,C 180.000} C_DIS
LIN {X 0.997,Y -28.996,Z -32.439,A 0.015,B -0.000,C 180.000} C_DIS
LIN {X 5.523,Y -24.191,Z -32.683,A 0.015,B 0.000,C 180.000} C_DIS
LIN {X 2.938,Y -18.117,Z -32.927,A 0.015,B 0.000,C -180.000} C_DIS
LIN {X -3.663,Y -18.047,Z -33.171,A 0.015,B 0.000,C 180.000} C_DIS
LIN {X -6.376,Y -24.064,Z -33.415,A 0.015,B -0.000,C 180.000} C_DIS
LIN {X -1.954,Y -28.964,Z -33.659,A 0.015,B 0.000,C 180.000} C_DIS
LIN {X 4.309,Y -26.881,Z -33.902,A 0.015,B 0.000,C -180.000} C_DIS
LIN {X 4.915,Y -20.308,Z -34.146,A 0.015,B 0.000,C 180.000} C_DIS
LIN {X -0.863,Y -17.115,Z -34.390,A 0.015,B 0.000,C -180.000} C_DIS
LIN {X -6.106,Y -21.126,Z -34.634,A 0.015,B 0.000,C -180.000} C_DIS
LIN {X -4.537,Y -27.537,Z -34.878,A 0.015,B 0.000,C -180.000} C_DIS
LIN {X 1.966,Y -28.674,Z -35.122,A 0.015,B 0.000,C 180.000} C_DIS
LIN {X 5.616,Y -23.174,Z -35.366,A 0.015,B 0.000,C 180.000} C_DIS
LIN {X 2.044,Y -17.623,Z -35.610,A 0.015,B 0.000,C 180.000} C_DIS
LIN {X -4.474,Y -18.667,Z -35.854,A 0.015,B 0.000,C -180.000} C_DIS
LIN {X -6.133,Y -25.056,Z -36.098,A 0.015,B 0.000,C 180.000} C_DIS
LIN {X -0.948,Y -29.140,Z -36.341,A 0.015,B 0.000,C 180.000} C_DIS
LIN {X 4.874,Y -26.030,Z -36.585,A 0.015,B 0.000,C 180.000} C_DIS
LIN {X 4.362,Y -19.449,Z -36.829,A 0.015,B 0.000,C 180.000} C_DIS
LIN {X -1.871,Y -17.277,Z -37.073,A 0.015,B 0.000,C 180.000} C_DIS
LIN {X -6.362,Y -22.114,Z -37.317,A 0.015,B 0.000,C 180.000} C_DIS
LIN {X -3.734,Y -28.169,Z -37.561,A 0.015,B 0.000,C 180.000} C_DIS
LIN {X 2.866,Y -28.192,Z -37.805,A 0.015,B -0.000,C -180.000} C_DIS
LIN {X 5.537,Y -22.156,Z -38.049,A 0.015,B 0.000,C -180.000} C_DIS
LIN {X 1.080,Y -17.287,Z -38.293,A 0.015,B 0.000,C -180.000} C_DIS
LIN {X -5.168,Y -19.415,Z -38.537,A 0.015,B 0.000,C -180.000} C_DIS
LIN {X -5.727,Y -25.993,Z -38.780,A 0.015,B 0.000,C -180.000} C_DIS
LIN {X 0.073,Y -29.144,Z -39.024,A 0.015,B 0.000,C -180.000} C_DIS
LIN {X 5.287,Y -25.096,Z -39.268,A 0.015,B 0.000,C 180.000} C_DIS
LIN {X 3.673,Y -18.696,Z -39.512,A 0.015,B 0.000,C -180.000} C_DIS
LIN {X -2.837,Y -17.606,Z -39.756,A 0.015,B 0.000,C 180.000} C_DIS
LIN {X -6.449,Y -23.131,Z -40.000,A 0.015,B 0.000,C 180.000} C_DIS
CIRC {X -0.842,Y -28.738,Z -40.000,A 0.015,B 0.000,C 180.000},{X 4.764,Y -23.131,Z -40.000,A 0.015,B 0.000,C 180.000} C_DIS
LIN {X 4.764,Y -20.362,Z -40.000,A 0.015,B -0.000,C -180.000} C_DIS
CIRC {X 3.658,Y -18.802,Z -40.000,A 0.015,B 0.000,C -180.000},{X 1.821,Y -19.329,Z -40.000,A 0.015,B 0.000,C 180.000} C_DIS
LIN {X -0.770,Y -22.568,Z -40.000,A 0.015,B -0.000,C -180.000} C_DIS
CIRC {X -1.006,Y -24.643,Z -40.000,A 0.015,B 0.000,C -180.000},{X 0.762,Y -25.755,Z -40.000,A 0.015,B 0.000,C -180.000} C_DIS
LIN {X 2.650,Y -25.755,Z -40.000,A 0.015,B 0.000,C 180.000} C_DIS
CIRC {X 4.145,Y -25.136,Z -40.000,A 0.015,B 0.000,C 180.000},{X 4.764,Y -23.641,Z -40.000,A 0.015,B 0.000,C 180.000} C_DIS
LIN {X 4.764,Y -23.131,Z -40.000,A 0.015,B -0.000,C -180.000} C_DIS
LIN {X 3.553,Y -23.398,Z -40.000,A 0.015,B 0.000,C 180.000} C_DIS
LIN {X 4.045,Y -24.462,Z -40.000,A 0.015,B 0.000,C 180.000} C_DIS
LIN {X 4.241,Y -24.704,Z -40.000,A 0.015,B 0.000,C -180.000} C_DIS
LIN {X 8.680,Y -28.027,Z -40.000,A 0.015,B 0.000,C -180.000} C_DIS
LIN {X 9.366,Y -28.668,Z -40.000,A 0.015,B -0.000,C -180.000} C_DIS
LIN {X 9.675,Y -28.604,Z -40.000,A 0.015,B -0.000,C 180.000} C_DIS
LIN {X 10.021,Y -27.803,Z -40.000,A 0.015,B 0.000,C 180.000} C_DIS
LIN {X 10.218,Y -26.938,Z -40.000,A 0.015,B -0.000,C 180.000} C_DIS
LIN {X 10.275,Y -25.867,Z -40.000,A 0.015,B 0.000,C 180.000} C_DIS
LIN {X 10.274,Y 7.442,Z -40.000,A 0.015,B 0.000,C 180.000} C_DIS
LIN {X 6.195,Y -2.894,Z -40.000,A 0.015,B 0.000,C 180.000} C_DIS
LIN {X 5.976,Y -3.347,Z -40.000,A 0.015,B 0.000,C 180.000} C_DIS
LIN {X 1.986,Y -10.239,Z -40.000,A 0.015,B 0.000,C -180.000} C_DIS
LIN {X 1.700,Y -10.657,Z -40.000,A 0.015,B 0.000,C 180.000} C_DIS
LIN {X -6.165,Y -20.492,Z -40.000,A 0.015,B 0.000,C 180.000} C_DIS
LIN {X -6.614,Y -20.955,Z -40.000,A 0.015,B -0.000,C 180.000} C_DIS
LIN {X -7.365,Y -21.594,Z -40.000,A 0.015,B 0.000,C -180.000} C_DIS
LIN {X -7.667,Y -21.823,Z -40.000,A 0.015,B -0.000,C -180.000} C_DIS
LIN {X -17.478,Y -28.433,Z -40.000,A 0.015,B 0.000,C 180.000} C_DIS
LIN {X -17.944,Y -28.696,Z -40.000,A 0.015,B 0.000,C -180.000} C_DIS
LIN {X -19.174,Y -29.267,Z -40.000,A 0.015,B 0.000,C 180.000} C_DIS
LIN {X -19.625,Y -29.438,Z -40.000,A 0.015,B -0.000,C -180.000} C_DIS
LIN {X -25.705,Y -31.266,Z -40.000,A 0.015,B 0.000,C 180.000} C_DIS
LIN {X 5.412,Y -31.266,Z -40.000,A 0.015,B 0.000,C -180.000} C_DIS
LIN {X 6.622,Y -31.073,Z -40.000,A 0.015,B 0.000,C 180.000} C_DIS
LIN {X 7.443,Y -30.763,Z -40.000,A 0.015,B 0.000,C 180.000} C_DIS
LIN {X 7.663,Y -30.627,Z -40.000,A 0.015,B 0.000,C -180.000} C_DIS
LIN {X 7.671,Y -29.553,Z -40.000,A 0.015,B 0.000,C -180.000} C_DIS
LIN {X 3.920,Y -27.149,Z -40.000,A 0.015,B 0.000,C -180.000} C_DIS
LIN {X -0.528,Y -24.823,Z -40.000,A 0.015,B 0.000,C 180.000} C_DIS
LIN {X -1.532,Y -24.257,Z -40.000,A 0.015,B 0.000,C -180.000} C_DIS
LIN {X -1.891,Y -24.456,Z -40.000,A 0.015,B -0.000,C 180.000} C_DIS
LIN {X 1.288,Y -30.046,Z -40.237,A 0.015,B 0.000,C 180.000} C_DIS
LIN {X 7.703,Y -29.592,Z -40.474,A 0.015,B -0.000,C 180.000} C_DIS
LIN {X 10.064,Y -23.611,Z -40.711,A 0.015,B 0.000,C 180.000} C_DIS
LIN {X 5.688,Y -18.898,Z -40.947,A 0.015,B 0.000,C 180.000} C_DIS
LIN {X -0.452,Y -20.810,Z -41.184,A 0.015,B 0.000,C 180.000} C_DIS
LIN {X -1.379,Y -27.173,Z -41.421,A 0.015,B -0.000,C 180.000} C_DIS
LIN {X 3.960,Y -30.757,Z -41.658,A 0.015,B 0.000,C 180.000} C_DIS
LIN {X 9.499,Y -27.489,Z -41.895,A 0.015,B 0.000,C -180.000} C_DIS
LIN {X 8.943,Y -21.083,Z -42.132,A 0.015,B 0.000,C 180.000} C_DIS
LIN {X 2.924,Y -18.818,Z -42.368,A 0.015,B 0.000,C 180.000} C_DIS
LIN {X -1.718,Y -23.268,Z -42.605,A 0.015,B 0.000,C -180.000} C_DIS
LIN {X 0.292,Y -29.377,Z -42.842,A 0.015,B 0.000,C 180.000} C_DIS
LIN {X 6.670,Y -30.202,Z -43.079,A 0.015,B 0.000,C -180.000} C_DIS
LIN {X 10.168,Y -24.806,Z -43.316,A 0.015,B 0.000,C 180.000} C_DIS
LIN {X 6.811,Y -19.321,Z -43.553,A 0.015,B 0.000,C -180.000} C_DIS
LIN {X 0.414,Y -19.980,Z -43.789,A 0.015,B 0.000,C 180.000} C_DIS
LIN {X -1.754,Y -26.034,Z -44.026,A 0.015,B -0.000,C -180.000} C_DIS
LIN {X 2.771,Y -30.603,Z -44.263,A 0.015,B 0.000,C 180.000} C_DIS
LIN {X 8.846,Y -28.496,Z -44.500,A 0.015,B -0.000,C -180.000} C_DIS
CIRC {X 7.971,Y -20.616,Z -44.500,A 0.015,B 0.000,C 180.000},{X 0.090,Y -21.491,Z -44.500,A 0.015,B 0.000,C -180.000} C_DIS
LIN {X -0.771,Y -22.568,Z -44.500,A 0.015,B 0.000,C 180.000} C_DIS
CIRC {X -1.007,Y -24.643,Z -44.500,A 0.015,B 0.000,C 180.000},{X 0.761,Y -25.755,Z -44.500,A 0.015,B -0.000,C 180.000} C_DIS
LIN {X 2.650,Y -25.755,Z -44.500,A 0.015,B -0.000,C 180.000} C_DIS
CIRC {X 4.145,Y -25.136,Z -44.500,A 0.015,B 0.000,C 180.000},{X 4.764,Y -23.641,Z -44.500,A 0.015,B -0.000,C 180.000} C_DIS
LIN {X 4.764,Y -20.362,Z -44.500,A 0.015,B 0.000,C -180.000} C_DIS
CIRC {X 3.658,Y -18.802,Z -44.500,A 0.015,B 0.000,C -180.000},{X 1.820,Y -19.329,Z -44.500,A 0.015,B 0.000,C 180.000} C_DIS
LIN {X 0.090,Y -21.491,Z -44.500,A 0.015,B 0.000,C -180.000} C_DIS
CIRC {X -0.123,Y -22.223,Z -44.500,A 0.015,B 0.000,C -180.000},{X 0.241,Y -22.892,Z -44.500,A 0.015,B 0.000,C -180.000} C_DIS
LIN {X 7.766,Y -29.001,Z -44.500,A 0.015,B 0.000,C -180.000} C_DIS
LIN {X 7.663,Y -30.627,Z -44.500,A 0.015,B 0.000,C 180.000} C_DIS
LIN {X 7.443,Y -30.763,Z -44.500,A 0.015,B 0.000,C 180.000} C_DIS
LIN {X 6.622,Y -31.073,Z -44.500,A 0.015,B 0.000,C -180.000} C_DIS
LIN {X 5.412,Y -31.266,Z -44.500,A 0.015,B -0.000,C 180.000} C_DIS
LIN {X -25.718,Y -31.266,Z -44.500,A 0.015,B 0.000,C -180.000} C_DIS
LIN {X -19.627,Y -29.439,Z -44.500,A 0.015,B 0.000,C -180.000} C_DIS
LIN {X -19.186,Y -29.273,Z -44.500,A 0.015,B 0.000,C -180.000} C_DIS
LIN {X -17.956,Y -28.707,Z -44.500,A 0.015,B 0.000,C 180.000} C_DIS
LIN {X -17.477,Y -28.438,Z -44.500,A 0.015,B 0.000,C -180.000} C_DIS
LIN {X -7.666,Y -21.822,Z -44.500,A 0.015,B -0.000,C -180.000} C_DIS
LIN {X -7.371,Y -21.599,Z -44.500,A 0.015,B -0.000,C 180.000} C_DIS
LIN {X -6.634,Y -20.974,Z -44.500,A 0.015,B 0.000,C 180.000} C_DIS
LIN {X -6.180,Y -20.507,Z -44.500,A 0.015,B 0.000,C -180.000} C_DIS
LIN {X 1.700,Y -10.657,Z -44.500,A 0.015,B 0.000,C -180.000} C_DIS
LIN {X 1.986,Y -10.239,Z -44.500,A 0.015,B 0.000,C -180.000} C_DIS
LIN {X 5.976,Y -3.347,Z -44.500,A 0.015,B -0.000,C 180.000} C_DIS
LIN {X 6.194,Y -2.895,Z -44.500,A 0.015,B 0.000,C 180.000} C_DIS
LIN {X 10.274,Y 7.429,Z -44.500,A 0.015,B 0.000,C -180.000} C_DIS
LIN {X 10.275,Y -25.867,Z -44.500,A 0.015,B -0.000,C 180.000} C_DIS
LIN {X 10.218,Y -26.938,Z -44.500,A 0.015,B 0.000,C 180.000} C_DIS
LIN {X 10.021,Y -27.803,Z -44.500,A 0.015,B 0.000,C -180.000} C_DIS
LIN {X 9.675,Y -28.604,Z -44.500,A 0.015,B 0.000,C 180.000} C_DIS
LIN {X 9.370,Y -28.671,Z -44.500,A 0.015,B 0.000,C 180.000} C_DIS
LIN {X 8.665,Y -28.047,Z -44.500,A 0.015,B 0.000,C 180.000} C_DIS
LIN {X 5.054,Y -25.579,Z -44.500,A 0.015,B -0.000,C 180.000} C_DIS
LIN {X 5.312,Y -26.059,Z -44.500,A 0.015,B 0.000,C 180.000} C_DIS
LIN {X 5.259,Y -25.177,Z -44.500,A 0.015,B 0.000,C 180.000} C_DIS
LIN {X 3.736,Y -18.755,Z -44.744,A 0.015,B 0.000,C 180.000} C_DIS
LIN {X -2.758,Y -17.572,Z -44.988,A 0.015,B -0.000,C 180.000} C_DIS
LIN {X -6.448,Y -23.046,Z -45.232,A 0.015,B -0.000,C 180.000} C_DIS
LIN {X -2.916,Y -28.622,Z -45.476,A 0.015,B 0.000,C 180.000} C_DIS
LIN {X 3.609,Y -27.624,Z -45.720,A 0.015,B -0.000,C 180.000} C_DIS
LIN {X 5.315,Y -21.248,Z -45.963,A 0.015,B 0.000,C -180.000} C_DIS
LIN {X 0.159,Y -17.126,Z -46.207,A 0.015,B 0.000,C -180.000} C_DIS
LIN {X -5.686,Y -20.195,Z -46.451,A 0.015,B -0.000,C -180.000} C_DIS
LIN {X -5.221,Y -26.779,Z -46.695,A 0.015,B 0.000,C 180.000} C_DIS
LIN {X 0.997,Y -28.996,Z -46.939,A 0.015,B -0.000,C 180.000} C_DIS
LIN {X 5.523,Y -24.191,Z -47.183,A 0.015,B 0.000,C 180.000} C_DIS
LIN {X 2.938,Y -18.117,Z -47.427,A 0.015,B 0.000,C -180.000} C_DIS
LIN {X -3.662,Y -18.047,Z -47.671,A 0.015,B 0.000,C 180.000} C_DIS
LIN {X -6.376,Y -24.064,Z -47.915,A 0.015,B 0.000,C -180.000} C_DIS
LIN {X -1.954,Y -28.965,Z -48.159,A 0.015,B -0.000,C 180.000} C_DIS
LIN {X 4.310,Y -26.881,Z -48.402,A 0.015,B 0.000,C 180.000} C_DIS
LIN {X 4.915,Y -20.308,Z -48.646,A 0.015,B -0.000,C 180.000} C_DIS
LIN {X -0.863,Y -17.115,Z -48.890,A 0.015,B 0.000,C 180.000} C_DIS
LIN {X -6.105,Y -21.126,Z -49.134,A 0.015,B 0.000,C -180.000} C_DIS
LIN {X -4.536,Y -27.537,Z -49.378,A 0.015,B 0.000,C -180.000} C_DIS
LIN {X 1.966,Y -28.674,Z -49.622,A 0.015,B -0.000,C 180.000} C_DIS
LIN {X 5.616,Y -23.174,Z -49.866,A 0.015,B 0.000,C -180.000} C_DIS
LIN {X 2.044,Y -17.623,Z -50.110,A 0.015,B 0.000,C -180.000} C_DIS
LIN {X -4.473,Y -18.667,Z -50.354,A 0.015,B 0.000,C -180.000} C_DIS
LIN {X -6.133,Y -25.056,Z -50.598,A 0.015,B 0.000,C -180.000} C_DIS
LIN {X -0.948,Y -29.140,Z -50.841,A 0.015,B 0.000,C -180.000} C_DIS
LIN {X 4.874,Y -26.030,Z -51.085,A 0.015,B 0.000,C 180.000} C_DIS
LIN {X 4.362,Y -19.449,Z -51.329,A 0.015,B 0.000,C -180.000} C_DIS
LIN {X -1.871,Y -17.277,Z -51.573,A 0.015,B 0.000,C 180.000} C_DIS
LIN {X -6.362,Y -22.114,Z -51.817,A 0.015,B 0.000,C 180.000} C_DIS
LIN {X -3.734,Y -28.169,Z -52.061,A 0.015,B 0.000,C 180.000} C_DIS
LIN {X 2.866,Y -28.193,Z -52.305,A 0.015,B 0.000,C 180.000} C_DIS
LIN {X 5.537,Y -22.156,Z -52.549,A 0.015,B 0.000,C 180.000} C_DIS
LIN {X 1.080,Y -17.287,Z -52.793,A 0.015,B 0.000,C 180.000} C_DIS
LIN {X -5.168,Y -19.416,Z -53.037,A 0.015,B 0.000,C 180.000} C_DIS
LIN {X -5.727,Y -25.993,Z -53.280,A 0.015,B -0.000,C -180.000} C_DIS
LIN {X 0.073,Y -29.144,Z -53.524,A 0.015,B 0.000,C 180.000} C_DIS
LIN {X 5.287,Y -25.096,Z -53.768,A 0.015,B 0.000,C -180.000} C_DIS
LIN {X 3.673,Y -18.696,Z -54.012,A 0.015,B -0.000,C 180.000} C_DIS
LIN {X -2.837,Y -17.606,Z -54.256,A 0.015,B 0.000,C -180.000} C_DIS
LIN {X -6.449,Y -23.132,Z -54.500,A 0.015,B -0.000,C 180.000} C_DIS
CIRC {X -0.842,Y -28.738,Z -54.500,A 0.015,B 0.000,C -180.000},{X 4.764,Y -23.131,Z -54.500,A 0.015,B -0.000,C -180.000} C_DIS
LIN {X 4.764,Y -20.362,Z -54.500,A 0.015,B -0.000,C -180.000} C_DIS
CIRC {X 3.658,Y -18.802,Z -54.500,A 0.015,B 0.000,C 180.000},{X 1.821,Y -19.329,Z -54.500,A 0.015,B 0.000,C -180.000} C_DIS
LIN {X -0.769,Y -22.568,Z -54.500,A 0.015,B 0.000,C 180.000} C_DIS
CIRC {X -1.005,Y -24.643,Z -54.500,A 0.015,B 0.000,C -180.000},{X 0.763,Y -25.755,Z -54.500,A 0.015,B 0.000,C -180.000} C_DIS
LIN {X 2.651,Y -25.755,Z -54.500,A 0.015,B 0.000,C -180.000} C_DIS
CIRC {X 4.145,Y -25.136,Z -54.500,A 0.015,B -0.000,C 180.000},{X 4.764,Y -23.641,Z -54.500,A 0.015,B 0.000,C -180.000} C_DIS
LIN {X 4.764,Y -23.131,Z -54.500,A 0.015,B -0.000,C -180.000} C_DIS
LIN {X 3.553,Y -23.398,Z -54.500,A 0.015,B 0.000,C -180.000} C_DIS
LIN {X 4.045,Y -24.462,Z -54.500,A 0.015,B -0.000,C 180.000} C_DIS
LIN {X 4.241,Y -24.704,Z -54.500,A 0.015,B 0.000,C 180.000} C_DIS
LIN {X 8.680,Y -28.027,Z -54.500,A 0.015,B 0.000,C 180.000} C_DIS
LIN {X 9.366,Y -28.668,Z -54.500,A 0.015,B 0.000,C -180.000} C_DIS
LIN {X 9.675,Y -28.604,Z -54.500,A 0.015,B 0.000,C 180.000} C_DIS
LIN {X 10.021,Y -27.803,Z -54.500,A 0.015,B 0.000,C 180.000} C_DIS
LIN {X 10.218,Y -26.938,Z -54.500,A 0.015,B 0.000,C 180.000} C_DIS
LIN {X 10.275,Y -25.867,Z -54.500,A 0.015,B 0.000,C 180.000} C_DIS
LIN {X 10.274,Y 7.407,Z -54.500,A 0.015,B -0.000,C 180.000} C_DIS
LIN {X 6.194,Y -2.898,Z -54.500,A 0.015,B -0.000,C -180.000} C_DIS
LIN {X 5.976,Y -3.347,Z -54.500,A 0.015,B 0.000,C 180.000} C_DIS
LIN {X 1.986,Y -10.239,Z -54.500,A 0.015,B -0.000,C -180.000} C_DIS
LIN {X 1.700,Y -10.657,Z -54.500,A 0.015,B -0.000,C 180.000} C_DIS
LIN {X -6.170,Y -20.499,Z -54.500,A 0.015,B -0.000,C 180.000} C_DIS
LIN {X -6.625,Y -20.967,Z -54.500,A 0.015,B 0.000,C -180.000} C_DIS
LIN {X -7.371,Y -21.598,Z -54.500,A 0.015,B -0.000,C 180.000} C_DIS
LIN {X -7.659,Y -21.817,Z -54.500,A 0.015,B 0.000,C 180.000} C_DIS
LIN {X -17.249,Y -28.322,Z -54.500,A 0.015,B 0.000,C 180.000} C_DIS
LIN {X -17.718,Y -28.588,Z -54.500,A 0.015,B 0.000,C -180.000} C_DIS
LIN {X -19.169,Y -29.265,Z -54.500,A 0.015,B 0.000,C 180.000} C_DIS
LIN {X -19.618,Y -29.436,Z -54.500,A 0.015,B 0.000,C -180.000} C_DIS
LIN {X -25.658,Y -31.266,Z -54.500,A 0.015,B -0.000,C -180.000} C_DIS
LIN {X 5.412,Y -31.266,Z -54.500,A 0.015,B -0.000,C 180.000} C_DIS
LIN {X 6.622,Y -31.073,Z -54.500,A 0.015,B -0.000,C -180.000} C_DIS
LIN {X 7.443,Y -30.763,Z -54.500,A 0.015,B -0.000,C 180.000} C_DIS
$VEL.CP = 1.00000
LIN {X 7.443,Y -30.763,Z 11.000,A 0.015,B 0.000,C 180.000} C_DIS
$VEL.CP = 1.00000
LIN {X 5.578,Y -23.911,Z 11.000,A 0.015,B 0.000,C 180.000} C_DIS
$VEL.CP = 0.10000
